Yaskawa INFORM job: DEMO_ROOF_SIDE_0625_3PAINT_26.JBI

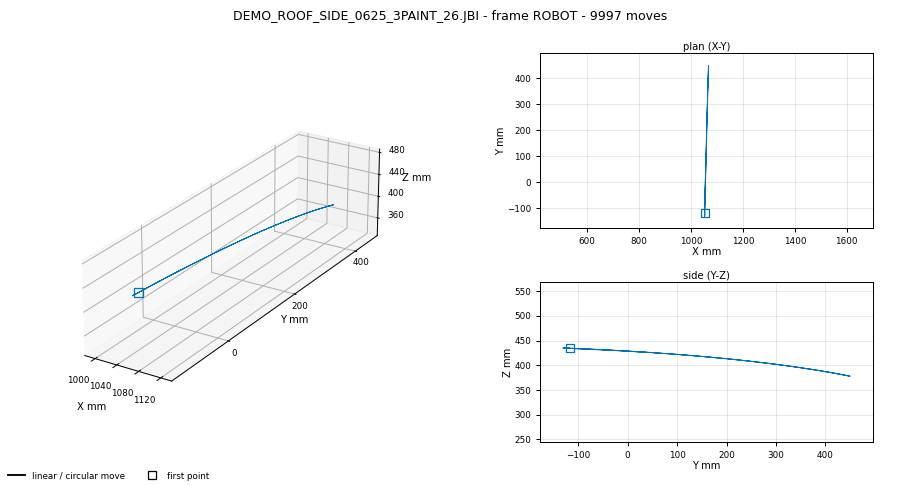
[picture p0: tool path of DEMO_ROOF_SIDE_0625_3PAINT_26.JBI in frame ROBOT, 9997 of 9997 moves have a stored position in this frame; points joined in program order, loops and branches not executed]
/JOB
//NAME DEMO_ROOF_SIDE_0625_3PAINT26
//POS
///NPOS 9997,0,0,0,0,0
///TOOL 0
///USER 0
///POSTYPE ROBOT
///RECTAN
///RCONF 1,0,0,0,0,0,0,0,0,0,0,0,0,0,0,0,0,0,0,0,0,0,0,0
C00000=1053.971,-116.920,435.028,170.360,28.855,155.473
C00001=1053.965,-117.170,435.037,170.358,28.855,155.473
C00002=1053.959,-117.419,435.047,170.356,28.854,155.473
C00003=1053.953,-117.669,435.057,170.354,28.853,155.473
C00004=1053.946,-117.919,435.066,170.352,28.853,155.473
C00005=1053.940,-118.169,435.076,170.349,28.852,155.473
C00006=1053.934,-118.419,435.084,170.347,28.852,155.474
C00007=1053.928,-118.669,435.094,170.345,28.851,155.474
C00008=1053.922,-118.918,435.103,170.343,28.851,155.474
C00009=1053.916,-119.168,435.112,170.341,28.850,155.474
C00010=1053.910,-119.417,435.122,170.339,28.850,155.474
C00011=1053.903,-119.667,435.131,170.337,28.849,155.474
C00012=1053.897,-119.917,435.141,170.335,28.849,155.474
C00013=1053.891,-120.167,435.151,170.333,28.848,155.474
C00014=1053.885,-120.417,435.160,170.331,28.847,155.474
C00015=1053.880,-120.666,435.169,170.329,28.847,155.474
C00016=1053.873,-120.916,435.178,170.327,28.847,155.474
C00017=1053.867,-121.166,435.187,170.324,28.846,155.474
C00018=1053.860,-121.415,435.197,170.322,28.846,155.474
C00019=1053.854,-121.665,435.206,170.320,28.845,155.475
C00020=1053.848,-121.915,435.216,170.319,28.845,155.475
C00021=1053.842,-122.165,435.225,170.317,28.844,155.475
C00022=1053.837,-122.414,435.234,170.315,28.844,155.475
C00023=1053.830,-122.664,435.243,170.312,28.843,155.475
C00024=1053.824,-122.914,435.252,170.310,28.843,155.475
C00025=1053.817,-123.164,435.262,170.308,28.842,155.475
C00026=1053.812,-123.414,435.271,170.306,28.842,155.475
C00027=1053.806,-123.663,435.280,170.304,28.842,155.475
C00028=1053.800,-123.913,435.290,170.302,28.841,155.475
C00029=1053.793,-124.162,435.299,170.299,28.841,155.475
C00030=1053.787,-124.413,435.307,170.297,28.840,155.476
C00031=1053.781,-124.663,435.317,170.295,28.840,155.476
C00032=1053.775,-124.912,435.326,170.294,28.840,155.476
C00033=1053.769,-125.162,435.334,170.292,28.839,155.476
C00034=1053.762,-125.412,435.344,170.290,28.839,155.476
C00035=1053.756,-125.661,435.354,170.287,28.838,155.476
C00036=1053.750,-125.911,435.363,170.285,28.838,155.476
C00037=1053.744,-126.161,435.371,170.283,28.838,155.476
C00038=1053.738,-126.410,435.381,170.281,28.838,155.476
C00039=1053.732,-126.660,435.390,170.279,28.837,155.477
C00040=1053.725,-126.910,435.398,170.276,28.837,155.477
C00041=1053.720,-127.159,435.408,170.274,28.836,155.477
C00042=1053.714,-127.410,435.417,170.272,28.836,155.477
C00043=1053.707,-127.659,435.425,170.271,28.835,155.477
C00044=1053.701,-127.909,435.436,170.269,28.835,155.477
C00045=1053.697,-128.159,435.445,170.267,28.835,155.477
C00046=1053.693,-128.409,435.455,170.265,28.833,155.477
C00047=1053.691,-128.659,435.466,170.263,28.831,155.477
C00048=1053.689,-128.909,435.479,170.262,28.828,155.476
C00049=1053.689,-129.161,435.491,170.260,28.825,155.476
C00050=1053.690,-129.411,435.503,170.259,28.822,155.475
C00051=1053.692,-129.660,435.518,170.258,28.818,155.475
C00052=1053.696,-129.912,435.532,170.257,28.813,155.474
C00053=1053.700,-130.163,435.547,170.256,28.808,155.473
C00054=1053.706,-130.413,435.563,170.256,28.802,155.472
C00055=1053.713,-130.663,435.580,170.256,28.796,155.471
C00056=1053.343,-130.687,435.365,170.208,28.964,155.504
C00057=1053.336,-130.437,435.348,170.208,28.970,155.505
C00058=1053.331,-130.186,435.333,170.209,28.975,155.506
C00059=1053.326,-129.936,435.318,170.210,28.981,155.507
C00060=1053.323,-129.684,435.303,170.210,28.985,155.508
C00061=1053.320,-129.434,435.290,170.212,28.989,155.508
C00062=1053.320,-129.183,435.276,170.213,28.993,155.509
C00063=1053.320,-128.933,435.264,170.214,28.996,155.509
C00064=1053.321,-128.683,435.251,170.216,28.998,155.510
C00065=1053.323,-128.432,435.240,170.218,29.001,155.510
C00066=1053.327,-128.182,435.230,170.219,29.002,155.510
C00067=1053.331,-127.932,435.220,170.221,29.003,155.510
C00068=1053.337,-127.682,435.211,170.223,29.004,155.510
C00069=1053.343,-127.433,435.202,170.225,29.004,155.510
C00070=1053.349,-127.183,435.193,170.227,29.004,155.510
C00071=1053.355,-126.933,435.184,170.230,29.004,155.510
C00072=1053.361,-126.683,435.174,170.232,29.005,155.509
C00073=1053.368,-126.434,435.166,170.234,29.005,155.509
C00074=1053.374,-126.184,435.157,170.236,29.006,155.509
C00075=1053.380,-125.934,435.147,170.237,29.006,155.509
C00076=1053.387,-125.685,435.138,170.240,29.006,155.509
C00077=1053.392,-125.435,435.130,170.242,29.006,155.509
C00078=1053.398,-125.185,435.120,170.244,29.007,155.509
C00079=1053.404,-124.935,435.111,170.246,29.007,155.509
C00080=1053.411,-124.686,435.102,170.248,29.008,155.509
C00081=1053.417,-124.435,435.093,170.251,29.008,155.509
C00082=1053.423,-124.186,435.084,170.253,29.009,155.508
C00083=1053.429,-123.937,435.074,170.255,29.009,155.508
C00084=1053.435,-123.686,435.066,170.257,29.010,155.508
C00085=1053.442,-123.437,435.056,170.259,29.010,155.508
C00086=1053.448,-123.187,435.047,170.261,29.010,155.508
C00087=1053.453,-122.938,435.037,170.264,29.010,155.508
C00088=1053.460,-122.688,435.028,170.265,29.011,155.508
C00089=1053.465,-122.438,435.019,170.267,29.011,155.508
C00090=1053.472,-122.188,435.010,170.269,29.012,155.508
C00091=1053.478,-121.938,435.000,170.271,29.012,155.508
C00092=1053.485,-121.688,434.991,170.273,29.012,155.507
C00093=1053.490,-121.439,434.982,170.276,29.013,155.507
C00094=1053.496,-121.189,434.973,170.278,29.013,155.507
C00095=1053.502,-120.939,434.963,170.280,29.014,155.507
C00096=1053.508,-120.689,434.954,170.282,29.014,155.507
C00097=1053.515,-120.440,434.945,170.284,29.015,155.507
C00098=1053.522,-120.190,434.935,170.285,29.016,155.507
C00099=1053.528,-119.940,434.926,170.288,29.016,155.507
C00100=1053.533,-119.691,434.916,170.290,29.017,155.507
C00101=1053.539,-119.441,434.908,170.292,29.017,155.507
C00102=1053.545,-119.191,434.898,170.294,29.018,155.507
C00103=1053.551,-118.941,434.888,170.296,29.018,155.507
C00104=1053.558,-118.691,434.879,170.299,29.019,155.507
C00105=1053.564,-118.442,434.869,170.301,29.019,155.506
C00106=1053.570,-118.192,434.860,170.303,29.019,155.506
C00107=1053.577,-117.942,434.851,170.305,29.020,155.506
C00108=1053.582,-117.693,434.842,170.307,29.020,155.506
C00109=1053.589,-117.443,434.832,170.308,29.021,155.506
C00110=1053.595,-117.194,434.822,170.311,29.022,155.506
C00111=1053.601,-116.944,434.813,170.313,29.022,155.506
C00112=1053.607,-116.694,434.803,170.315,29.023,155.506
C00113=1053.613,-116.444,434.794,170.317,29.023,155.506
C00114=1053.620,-116.194,434.784,170.319,29.024,155.506
C00115=1053.626,-115.945,434.775,170.321,29.024,155.506
C00116=1053.632,-115.695,434.765,170.324,29.025,155.506
C00117=1053.638,-115.411,434.755,170.326,29.026,155.506
C00118=1053.646,-115.126,434.743,170.328,29.026,155.505
C00119=1053.653,-114.841,434.733,170.330,29.027,155.505
C00120=1053.660,-114.558,434.722,170.332,29.027,155.505
C00121=1053.666,-114.308,434.712,170.335,29.028,155.505
C00122=1053.672,-114.058,434.703,170.337,29.029,155.505
C00123=1053.678,-113.808,434.693,170.339,29.029,155.505
C00124=1053.684,-113.558,434.683,170.341,29.030,155.505
C00125=1053.690,-113.308,434.673,170.343,29.031,155.505
C00126=1053.696,-113.059,434.664,170.345,29.031,155.505
C00127=1053.702,-112.809,434.654,170.348,29.032,155.505
C00128=1053.709,-112.559,434.645,170.349,29.033,155.505
C00129=1053.715,-112.309,434.635,170.351,29.033,155.505
C00130=1053.721,-112.059,434.626,170.353,29.033,155.505
C00131=1053.727,-111.810,434.615,170.355,29.034,155.505
C00132=1053.734,-111.560,434.606,170.357,29.035,155.505
C00133=1053.740,-111.311,434.596,170.360,29.035,155.505
C00134=1053.746,-111.061,434.587,170.362,29.037,155.505
C00135=1053.751,-110.811,434.576,170.364,29.037,155.505
C00136=1053.757,-110.561,434.567,170.366,29.037,155.504
C00137=1053.764,-110.312,434.557,170.367,29.038,155.505
C00138=1053.770,-110.062,434.547,170.369,29.039,155.504
C00139=1053.776,-109.812,434.537,170.372,29.039,155.504
C00140=1053.782,-109.562,434.528,170.374,29.040,155.504
C00141=1053.789,-109.313,434.518,170.376,29.041,155.504
C00142=1053.795,-109.063,434.508,170.378,29.041,155.504
C00143=1053.801,-108.814,434.498,170.380,29.042,155.504
C00144=1053.807,-108.563,434.488,170.382,29.043,155.504
C00145=1053.813,-108.314,434.479,170.384,29.044,155.504
C00146=1053.819,-108.064,434.469,170.386,29.044,155.504
C00147=1053.826,-107.815,434.459,170.388,29.045,155.504
C00148=1053.832,-107.565,434.449,170.390,29.046,155.504
C00149=1053.838,-107.315,434.440,170.392,29.046,155.504
C00150=1053.844,-107.066,434.429,170.394,29.047,155.504
C00151=1053.850,-106.816,434.419,170.397,29.048,155.504
C00152=1053.856,-106.566,434.410,170.399,29.049,155.504
C00153=1053.862,-106.316,434.400,170.400,29.049,155.504
C00154=1053.869,-106.066,434.389,170.402,29.050,155.504
C00155=1053.875,-105.816,434.379,170.404,29.051,155.504
C00156=1053.881,-105.566,434.370,170.406,29.052,155.504
C00157=1053.887,-105.317,434.359,170.409,29.052,155.504
C00158=1053.893,-105.067,434.349,170.411,29.053,155.504
C00159=1053.899,-104.817,434.340,170.413,29.054,155.504
C00160=1053.905,-104.568,434.329,170.415,29.055,155.504
C00161=1053.912,-104.318,434.320,170.416,29.056,155.504
C00162=1053.917,-104.069,434.309,170.418,29.056,155.504
C00163=1053.923,-103.819,434.299,170.420,29.057,155.504
C00164=1053.930,-103.569,434.290,170.423,29.058,155.504
C00165=1053.936,-103.319,434.279,170.425,29.059,155.504
C00166=1053.942,-103.069,434.269,170.427,29.060,155.504
C00167=1053.949,-102.820,434.259,170.429,29.060,155.504
C00168=1053.954,-102.570,434.249,170.431,29.061,155.504
C00169=1053.960,-102.320,434.239,170.432,29.062,155.503
C00170=1053.967,-102.071,434.229,170.434,29.063,155.503
C00171=1053.972,-101.821,434.219,170.437,29.064,155.503
C00172=1053.979,-101.572,434.208,170.439,29.064,155.503
C00173=1053.985,-101.321,434.198,170.441,29.065,155.503
C00174=1053.991,-101.072,434.188,170.443,29.066,155.503
C00175=1053.997,-100.822,434.178,170.445,29.067,155.503
C00176=1054.004,-100.573,434.168,170.446,29.068,155.503
C00177=1054.009,-100.323,434.158,170.449,29.069,155.503
C00178=1054.016,-100.073,434.147,170.451,29.069,155.503
C00179=1054.022,-99.823,434.137,170.453,29.070,155.503
C00180=1054.028,-99.573,434.126,170.455,29.072,155.503
C00181=1054.035,-99.287,434.115,170.457,29.072,155.503
C00182=1054.042,-99.001,434.103,170.460,29.073,155.503
C00183=1054.050,-98.716,434.092,170.461,29.074,155.503
C00184=1054.057,-98.431,434.080,170.464,29.075,155.503
C00185=1054.063,-98.180,434.070,170.466,29.076,155.503
C00186=1054.069,-97.931,434.060,170.468,29.077,155.503
C00187=1054.075,-97.682,434.049,170.470,29.078,155.503
C00188=1054.081,-97.432,434.039,170.472,29.079,155.503
C00189=1054.087,-97.182,434.028,170.475,29.079,155.503
C00190=1054.094,-96.932,434.018,170.476,29.080,155.503
C00191=1054.099,-96.682,434.007,170.478,29.082,155.503
C00192=1054.106,-96.433,433.997,170.480,29.083,155.503
C00193=1054.111,-96.183,433.987,170.482,29.084,155.503
C00194=1054.118,-95.934,433.977,170.484,29.085,155.503
C00195=1054.124,-95.684,433.965,170.486,29.086,155.503
C00196=1054.130,-95.434,433.955,170.488,29.087,155.504
C00197=1054.136,-95.184,433.945,170.490,29.088,155.503
C00198=1054.142,-94.935,433.934,170.492,29.088,155.503
C00199=1054.148,-94.685,433.925,170.494,29.089,155.503
C00200=1054.154,-94.435,433.913,170.496,29.090,155.503
C00201=1054.160,-94.186,433.902,170.498,29.091,155.504
C00202=1054.167,-93.936,433.892,170.500,29.092,155.504
C00203=1054.172,-93.686,433.882,170.502,29.093,155.504
C00204=1054.179,-93.436,433.871,170.504,29.095,155.504
C00205=1054.185,-93.187,433.860,170.506,29.096,155.504
C00206=1054.190,-92.937,433.850,170.508,29.097,155.504
C00207=1054.197,-92.688,433.840,170.510,29.098,155.504
C00208=1054.203,-92.437,433.829,170.512,29.099,155.504
C00209=1054.209,-92.188,433.818,170.514,29.100,155.504
C00210=1054.215,-91.939,433.808,170.515,29.101,155.504
C00211=1054.221,-91.689,433.797,170.517,29.102,155.504
C00212=1054.228,-91.439,433.787,170.520,29.103,155.504
C00213=1054.233,-91.189,433.776,170.522,29.104,155.504
C00214=1054.239,-90.940,433.765,170.524,29.105,155.504
C00215=1054.246,-90.690,433.754,170.526,29.106,155.504
C00216=1054.252,-90.440,433.744,170.527,29.107,155.504
C00217=1054.257,-90.190,433.733,170.529,29.108,155.504
C00218=1054.264,-89.941,433.723,170.531,29.109,155.504
C00219=1054.270,-89.691,433.712,170.533,29.110,155.504
C00220=1054.276,-89.441,433.701,170.536,29.111,155.504
C00221=1054.282,-89.192,433.691,170.538,29.112,155.504
C00222=1054.289,-88.942,433.679,170.540,29.113,155.504
C00223=1054.295,-88.692,433.670,170.541,29.114,155.504
C00224=1054.301,-88.443,433.659,170.543,29.115,155.504
C00225=1054.307,-88.193,433.648,170.545,29.116,155.504
C00226=1054.314,-87.943,433.637,170.547,29.117,155.504
C00227=1054.319,-87.694,433.627,170.549,29.118,155.504
C00228=1054.326,-87.444,433.615,170.552,29.120,155.504
C00229=1054.332,-87.195,433.605,170.553,29.121,155.504
C00230=1054.338,-86.944,433.594,170.555,29.122,155.504
C00231=1054.344,-86.695,433.583,170.557,29.123,155.504
C00232=1054.351,-86.446,433.573,170.559,29.124,155.504
C00233=1054.357,-86.195,433.561,170.561,29.125,155.504
C00234=1054.363,-85.946,433.550,170.563,29.126,155.505
C00235=1054.369,-85.696,433.540,170.565,29.127,155.505
C00236=1054.376,-85.447,433.529,170.567,29.129,155.505
C00237=1054.381,-85.197,433.518,170.569,29.130,155.505
C00238=1054.388,-84.947,433.507,170.571,29.131,155.505
C00239=1054.394,-84.698,433.497,170.573,29.132,155.505
C00240=1054.400,-84.448,433.485,170.575,29.133,155.505
C00241=1054.406,-84.198,433.474,170.577,29.134,155.505
C00242=1054.413,-83.949,433.464,170.578,29.135,155.505
C00243=1054.419,-83.699,433.453,170.580,29.136,155.505
C00244=1054.425,-83.449,433.442,170.583,29.137,155.505
C00245=1054.432,-83.165,433.429,170.585,29.139,155.505
C00246=1054.439,-82.882,433.418,170.587,29.140,155.505
C00247=1054.446,-82.598,433.405,170.589,29.141,155.505
C00248=1054.454,-82.315,433.392,170.591,29.142,155.505
C00249=1054.460,-82.066,433.381,170.593,29.143,155.505
C00250=1054.466,-81.815,433.370,170.595,29.144,155.505
C00251=1054.472,-81.566,433.359,170.597,29.145,155.505
C00252=1054.479,-81.316,433.349,170.600,29.147,155.505
C00253=1054.485,-81.067,433.338,170.601,29.148,155.505
C00254=1054.491,-80.816,433.327,170.603,29.149,155.506
C00255=1054.497,-80.567,433.316,170.605,29.150,155.506
C00256=1054.504,-80.317,433.305,170.607,29.151,155.506
C00257=1054.510,-80.068,433.293,170.609,29.152,155.506
C00258=1054.516,-79.818,433.282,170.611,29.153,155.506
C00259=1054.522,-79.568,433.271,170.612,29.155,155.506
C00260=1054.528,-79.318,433.260,170.614,29.156,155.506
C00261=1054.534,-79.069,433.249,170.617,29.157,155.506
C00262=1054.540,-78.820,433.238,170.619,29.159,155.506
C00263=1054.546,-78.570,433.226,170.621,29.160,155.506
C00264=1054.552,-78.320,433.215,170.623,29.161,155.506
C00265=1054.559,-78.070,433.205,170.624,29.162,155.506
C00266=1054.565,-77.821,433.193,170.626,29.163,155.506
C00267=1054.572,-77.571,433.182,170.628,29.165,155.506
C00268=1054.577,-77.322,433.171,170.630,29.166,155.506
C00269=1054.584,-77.072,433.160,170.632,29.167,155.506
C00270=1054.590,-76.823,433.148,170.633,29.169,155.507
C00271=1054.596,-76.573,433.137,170.636,29.170,155.507
C00272=1054.602,-76.323,433.126,170.638,29.172,155.507
C00273=1054.608,-76.073,433.115,170.640,29.173,155.507
C00274=1054.615,-75.823,433.103,170.642,29.174,155.507
C00275=1054.621,-75.574,433.092,170.644,29.175,155.507
C00276=1054.627,-75.324,433.081,170.645,29.176,155.507
C00277=1054.633,-75.075,433.069,170.647,29.178,155.507
C00278=1054.639,-74.825,433.058,170.649,29.179,155.507
C00279=1054.645,-74.575,433.047,170.651,29.180,155.507
C00280=1054.652,-74.325,433.035,170.653,29.182,155.507
C00281=1054.657,-74.076,433.024,170.656,29.183,155.507
C00282=1054.664,-73.826,433.012,170.657,29.184,155.508
C00283=1054.670,-73.577,433.001,170.659,29.185,155.508
C00284=1054.675,-73.326,432.990,170.661,29.187,155.508
C00285=1054.682,-73.077,432.978,170.663,29.189,155.508
C00286=1054.688,-72.827,432.967,170.665,29.190,155.508
C00287=1054.694,-72.578,432.955,170.666,29.191,155.508
C00288=1054.700,-72.328,432.944,170.668,29.192,155.508
C00289=1054.706,-72.078,432.932,170.670,29.194,155.508
C00290=1054.712,-71.829,432.920,170.672,29.195,155.508
C00291=1054.718,-71.579,432.909,170.674,29.196,155.508
C00292=1054.724,-71.330,432.898,170.675,29.198,155.509
C00293=1054.730,-71.079,432.886,170.677,29.199,155.509
C00294=1054.736,-70.830,432.874,170.679,29.201,155.509
C00295=1054.742,-70.580,432.863,170.682,29.203,155.509
C00296=1054.749,-70.331,432.851,170.684,29.204,155.509
C00297=1054.754,-70.081,432.840,170.685,29.205,155.509
C00298=1054.761,-69.831,432.828,170.687,29.207,155.509
C00299=1054.766,-69.582,432.817,170.689,29.208,155.509
C00300=1054.773,-69.332,432.805,170.691,29.209,155.509
C00301=1054.778,-69.082,432.793,170.693,29.211,155.510
C00302=1054.785,-68.833,432.781,170.695,29.212,155.510
C00303=1054.791,-68.583,432.769,170.696,29.214,155.510
C00304=1054.797,-68.334,432.758,170.698,29.215,155.510
C00305=1054.803,-68.084,432.746,170.700,29.216,155.510
C00306=1054.809,-67.834,432.735,170.702,29.218,155.510
C00307=1054.815,-67.585,432.723,170.704,29.220,155.510
C00308=1054.822,-67.335,432.712,170.705,29.221,155.510
C00309=1054.828,-67.054,432.698,170.708,29.222,155.510
C00310=1054.835,-66.773,432.684,170.710,29.224,155.511
C00311=1054.842,-66.492,432.672,170.712,29.226,155.511
C00312=1054.849,-66.210,432.658,170.714,29.227,155.511
C00313=1054.855,-65.960,432.647,170.716,29.229,155.511
C00314=1054.861,-65.711,432.635,170.718,29.230,155.511
C00315=1054.867,-65.461,432.623,170.720,29.232,155.511
C00316=1054.873,-65.211,432.612,170.722,29.233,155.511
C00317=1054.880,-64.962,432.600,170.723,29.235,155.511
C00318=1054.886,-64.712,432.587,170.725,29.236,155.511
C00319=1054.891,-64.462,432.576,170.727,29.238,155.512
C00320=1054.898,-64.213,432.564,170.729,29.239,155.512
C00321=1054.905,-63.963,432.552,170.731,29.241,155.512
C00322=1054.910,-63.713,432.541,170.732,29.242,155.512
C00323=1054.916,-63.464,432.529,170.734,29.243,155.512
C00324=1054.923,-63.214,432.517,170.736,29.245,155.512
C00325=1054.929,-62.964,432.504,170.739,29.247,155.512
C00326=1054.935,-62.715,432.494,170.741,29.248,155.512
C00327=1054.941,-62.465,432.482,170.742,29.249,155.513
C00328=1054.947,-62.215,432.469,170.744,29.251,155.513
C00329=1054.954,-61.966,432.457,170.746,29.253,155.513
C00330=1054.960,-61.716,432.446,170.748,29.254,155.513
C00331=1054.965,-61.466,432.434,170.750,29.255,155.513
C00332=1054.972,-61.217,432.422,170.751,29.257,155.513
C00333=1054.979,-60.967,432.410,170.753,29.259,155.513
C00334=1054.984,-60.718,432.398,170.755,29.260,155.514
C00335=1054.990,-60.468,432.386,170.757,29.261,155.514
C00336=1054.997,-60.218,432.374,170.759,29.263,155.514
C00337=1055.003,-59.968,432.362,170.760,29.264,155.514
C00338=1055.009,-59.720,432.350,170.762,29.266,155.514
C00339=1055.016,-59.470,432.338,170.764,29.268,155.514
C00340=1055.022,-59.220,432.326,170.766,29.269,155.514
C00341=1055.028,-58.970,432.314,170.768,29.270,155.514
C00342=1055.035,-58.720,432.302,170.769,29.272,155.515
C00343=1055.040,-58.471,432.290,170.772,29.274,155.515
C00344=1055.046,-58.222,432.278,170.774,29.275,155.515
C00345=1055.052,-57.972,432.266,170.776,29.277,155.515
C00346=1055.059,-57.722,432.254,170.778,29.278,155.515
C00347=1055.066,-57.473,432.242,170.779,29.279,155.515
C00348=1055.072,-57.223,432.229,170.781,29.281,155.515
C00349=1055.078,-56.974,432.218,170.783,29.283,155.515
C00350=1055.084,-56.724,432.206,170.785,29.284,155.516
C00351=1055.090,-56.474,432.193,170.787,29.286,155.516
C00352=1055.097,-56.224,432.182,170.788,29.287,155.516
C00353=1055.102,-55.974,432.169,170.790,29.289,155.516
C00354=1055.109,-55.725,432.157,170.792,29.290,155.516
C00355=1055.116,-55.475,432.145,170.794,29.292,155.516
C00356=1055.122,-55.225,432.133,170.796,29.293,155.516
C00357=1055.128,-54.976,432.121,170.797,29.295,155.517
C00358=1055.134,-54.726,432.109,170.799,29.297,155.517
C00359=1055.140,-54.477,432.097,170.801,29.298,155.517
C00360=1055.147,-54.227,432.085,170.803,29.299,155.517
C00361=1055.153,-53.977,432.072,170.805,29.301,155.517
C00362=1055.159,-53.728,432.060,170.806,29.302,155.517
C00363=1055.165,-53.478,432.048,170.808,29.304,155.517
C00364=1055.172,-53.228,432.036,170.810,29.306,155.517
C00365=1055.179,-52.979,432.024,170.812,29.307,155.518
C00366=1055.185,-52.730,432.011,170.814,29.309,155.518
C00367=1055.192,-52.480,431.999,170.815,29.310,155.518
C00368=1055.197,-52.231,431.986,170.818,29.312,155.518
C00369=1055.203,-51.981,431.975,170.820,29.314,155.518
C00370=1055.209,-51.731,431.962,170.822,29.315,155.518
C00371=1055.216,-51.482,431.950,170.824,29.316,155.518
C00372=1055.223,-51.232,431.938,170.825,29.318,155.519
C00373=1055.229,-50.952,431.924,170.827,29.320,155.519
C00374=1055.237,-50.672,431.910,170.829,29.322,155.519
C00375=1055.244,-50.392,431.897,170.831,29.324,155.519
C00376=1055.251,-50.112,431.882,170.833,29.325,155.519
C00377=1055.257,-49.862,431.869,170.835,29.327,155.519
C00378=1055.263,-49.612,431.857,170.837,29.329,155.520
C00379=1055.269,-49.363,431.845,170.839,29.331,155.520
C00380=1055.275,-49.113,431.833,170.841,29.332,155.520
C00381=1055.281,-48.864,431.820,170.842,29.334,155.520
C00382=1055.287,-48.614,431.807,170.844,29.336,155.520
C00383=1055.294,-48.365,431.795,170.846,29.337,155.520
C00384=1055.300,-48.115,431.782,170.848,29.339,155.521
C00385=1055.306,-47.865,431.770,170.849,29.341,155.521
C00386=1055.312,-47.616,431.756,170.851,29.343,155.521
C00387=1055.318,-47.366,431.745,170.853,29.344,155.521
C00388=1055.324,-47.116,431.732,170.855,29.346,155.521
C00389=1055.330,-46.866,431.719,170.857,29.347,155.521
C00390=1055.336,-46.617,431.706,170.858,29.349,155.522
C00391=1055.343,-46.368,431.694,170.860,29.351,155.522
C00392=1055.349,-46.118,431.682,170.862,29.353,155.522
C00393=1055.355,-45.868,431.668,170.864,29.354,155.522
C00394=1055.361,-45.619,431.656,170.866,29.356,155.522
C00395=1055.368,-45.369,431.644,170.867,29.358,155.522
C00396=1055.374,-45.120,431.631,170.869,29.360,155.523
C00397=1055.380,-44.870,431.618,170.871,29.361,155.523
C00398=1055.386,-44.620,431.605,170.873,29.363,155.523
C00399=1055.393,-44.371,431.593,170.874,29.365,155.523
C00400=1055.399,-44.121,431.580,170.876,29.366,155.523
C00401=1055.405,-43.871,431.568,170.878,29.369,155.524
C00402=1055.411,-43.622,431.554,170.880,29.370,155.524
C00403=1055.417,-43.372,431.542,170.882,29.372,155.524
C00404=1055.423,-43.122,431.530,170.883,29.373,155.524
C00405=1055.430,-42.873,431.517,170.885,29.376,155.524
C00406=1055.435,-42.623,431.504,170.887,29.377,155.525
C00407=1055.442,-42.374,431.491,170.889,29.379,155.525
C00408=1055.448,-42.124,431.478,170.890,29.380,155.525
C00409=1055.455,-41.875,431.466,170.892,29.382,155.525
C00410=1055.460,-41.625,431.453,170.894,29.384,155.525
C00411=1055.466,-41.375,431.440,170.896,29.386,155.525
C00412=1055.473,-41.126,431.427,170.898,29.387,155.526
C00413=1055.478,-40.876,431.415,170.899,29.389,155.526
C00414=1055.485,-40.627,431.402,170.901,29.391,155.526
C00415=1055.491,-40.377,431.389,170.903,29.393,155.526
C00416=1055.498,-40.128,431.376,170.905,29.394,155.526
C00417=1055.503,-39.878,431.364,170.906,29.396,155.526
C00418=1055.510,-39.628,431.350,170.908,29.398,155.527
C00419=1055.516,-39.378,431.337,170.910,29.400,155.527
C00420=1055.523,-39.130,431.325,170.912,29.401,155.527
C00421=1055.529,-38.880,431.312,170.914,29.404,155.527
C00422=1055.535,-38.630,431.299,170.915,29.405,155.527
C00423=1055.541,-38.380,431.286,170.917,29.407,155.528
C00424=1055.547,-38.131,431.273,170.919,29.409,155.528
C00425=1055.553,-37.881,431.261,170.921,29.411,155.528
C00426=1055.560,-37.632,431.247,170.922,29.412,155.528
C00427=1055.566,-37.383,431.234,170.923,29.414,155.528
C00428=1055.572,-37.133,431.221,170.925,29.416,155.529
C00429=1055.578,-36.883,431.208,170.927,29.418,155.529
C00430=1055.584,-36.633,431.195,170.929,29.420,155.529
C00431=1055.591,-36.384,431.182,170.930,29.422,155.529
C00432=1055.596,-36.134,431.168,170.932,29.423,155.529
C00433=1055.602,-35.884,431.156,170.934,29.425,155.530
C00434=1055.608,-35.635,431.142,170.936,29.427,155.530
C00435=1055.614,-35.386,431.129,170.937,29.429,155.530
C00436=1055.620,-35.136,431.116,170.939,29.431,155.530
C00437=1055.627,-34.856,431.102,170.941,29.433,155.530
C00438=1055.634,-34.577,431.087,170.944,29.435,155.531
C00439=1055.641,-34.297,431.072,170.945,29.437,155.531
C00440=1055.648,-34.018,431.058,170.947,29.439,155.531
C00441=1055.654,-33.768,431.044,170.949,29.441,155.531
C00442=1055.660,-33.518,431.031,170.951,29.443,155.532
C00443=1055.667,-33.269,431.018,170.952,29.445,155.532
C00444=1055.673,-33.019,431.005,170.954,29.446,155.532
C00445=1055.679,-32.770,430.991,170.956,29.449,155.532
C00446=1055.685,-32.520,430.979,170.958,29.450,155.532
C00447=1055.692,-32.270,430.965,170.960,29.452,155.533
C00448=1055.698,-32.021,430.952,170.961,29.454,155.533
C00449=1055.704,-31.772,430.939,170.963,29.456,155.533
C00450=1055.710,-31.522,430.926,170.965,29.458,155.533
C00451=1055.716,-31.273,430.913,170.966,29.460,155.534
C00452=1055.723,-31.023,430.899,170.967,29.461,155.534
C00453=1055.729,-30.773,430.885,170.969,29.464,155.534
C00454=1055.735,-30.524,430.872,170.971,29.465,155.534
C00455=1055.741,-30.274,430.860,170.973,29.467,155.534
C00456=1055.748,-30.024,430.846,170.975,29.469,155.535
C00457=1055.754,-29.775,430.833,170.976,29.471,155.535
C00458=1055.760,-29.525,430.819,170.978,29.473,155.535
C00459=1055.766,-29.276,430.806,170.980,29.475,155.535
C00460=1055.772,-29.027,430.793,170.982,29.477,155.535
C00461=1055.779,-28.776,430.780,170.983,29.479,155.536
C00462=1055.784,-28.527,430.766,170.985,29.480,155.536
C00463=1055.791,-28.277,430.753,170.987,29.483,155.536
C00464=1055.797,-28.027,430.739,170.989,29.484,155.536
C00465=1055.804,-27.778,430.726,170.990,29.486,155.537
C00466=1055.810,-27.529,430.713,170.992,29.488,155.537
C00467=1055.816,-27.280,430.699,170.994,29.490,155.537
C00468=1055.823,-27.030,430.686,170.996,29.492,155.537
C00469=1055.828,-26.780,430.672,170.997,29.494,155.537
C00470=1055.835,-26.531,430.659,170.998,29.495,155.538
C00471=1055.840,-26.281,430.646,171.000,29.498,155.538
C00472=1055.847,-26.031,430.632,171.002,29.500,155.538
C00473=1055.853,-25.781,430.618,171.004,29.501,155.538
C00474=1055.859,-25.532,430.605,171.005,29.504,155.539
C00475=1055.864,-25.283,430.591,171.007,29.506,155.539
C00476=1055.871,-25.033,430.578,171.009,29.507,155.539
C00477=1055.877,-24.783,430.564,171.011,29.509,155.539
C00478=1055.883,-24.534,430.551,171.012,29.512,155.540
C00479=1055.890,-24.284,430.537,171.014,29.513,155.540
C00480=1055.896,-24.035,430.524,171.016,29.515,155.540
C00481=1055.901,-23.785,430.510,171.018,29.518,155.540
C00482=1055.908,-23.536,430.497,171.019,29.519,155.540
C00483=1055.915,-23.286,430.482,171.020,29.521,155.541
C00484=1055.920,-23.037,430.468,171.022,29.523,155.541
C00485=1055.926,-22.788,430.455,171.024,29.525,155.541
C00486=1055.933,-22.537,430.441,171.026,29.527,155.541
C00487=1055.939,-22.288,430.428,171.027,29.529,155.542
C00488=1055.945,-22.039,430.414,171.029,29.531,155.542
C00489=1055.951,-21.788,430.400,171.031,29.533,155.542
C00490=1055.957,-21.539,430.387,171.033,29.535,155.542
C00491=1055.963,-21.290,430.374,171.034,29.537,155.543
C00492=1055.970,-21.040,430.359,171.036,29.539,155.543
C00493=1055.976,-20.790,430.346,171.038,29.541,155.543
C00494=1055.982,-20.541,430.331,171.040,29.544,155.543
C00495=1055.988,-20.291,430.318,171.040,29.545,155.544
C00496=1055.995,-20.042,430.305,171.042,29.547,155.544
C00497=1056.000,-19.793,430.291,171.044,29.549,155.544
C00498=1056.007,-19.543,430.277,171.046,29.551,155.544
C00499=1056.012,-19.293,430.263,171.047,29.553,155.545
C00500=1056.019,-19.044,430.249,171.049,29.555,155.545
C00501=1056.026,-18.763,430.233,171.051,29.558,155.545
C00502=1056.033,-18.483,430.219,171.053,29.560,155.545
C00503=1056.040,-18.202,430.203,171.054,29.562,155.546
C00504=1056.047,-17.923,430.187,171.057,29.564,155.546
C00505=1056.053,-17.672,430.173,171.058,29.566,155.546
C00506=1056.059,-17.423,430.160,171.060,29.568,155.546
C00507=1056.065,-17.174,430.145,171.061,29.570,155.547
C00508=1056.072,-16.924,430.132,171.063,29.572,155.547
C00509=1056.078,-16.675,430.118,171.065,29.574,155.547
C00510=1056.084,-16.425,430.104,171.067,29.576,155.547
C00511=1056.091,-16.176,430.090,171.069,29.578,155.548
C00512=1056.097,-15.926,430.076,171.070,29.580,155.548
C00513=1056.103,-15.676,430.063,171.072,29.582,155.548
C00514=1056.109,-15.427,430.049,171.074,29.584,155.548
C00515=1056.116,-15.178,430.035,171.075,29.586,155.549
C00516=1056.121,-14.928,430.021,171.076,29.588,155.549
C00517=1056.128,-14.678,430.007,171.078,29.591,155.549
C00518=1056.134,-14.429,429.992,171.080,29.593,155.549
C00519=1056.140,-14.179,429.978,171.082,29.594,155.550
C00520=1056.146,-13.930,429.965,171.083,29.596,155.550
C00521=1056.152,-13.681,429.950,171.085,29.599,155.550
C00522=1056.158,-13.430,429.936,171.087,29.601,155.550
C00523=1056.165,-13.182,429.922,171.089,29.603,155.551
C00524=1056.171,-12.931,429.908,171.089,29.605,155.551
C00525=1056.176,-12.682,429.894,171.091,29.607,155.551
C00526=1056.183,-12.432,429.880,171.093,29.609,155.551
C00527=1056.189,-12.183,429.866,171.095,29.611,155.552
C00528=1056.194,-11.934,429.851,171.096,29.613,155.552
C00529=1056.201,-11.684,429.838,171.098,29.615,155.552
C00530=1056.207,-11.434,429.824,171.100,29.618,155.552
C00531=1056.213,-11.185,429.809,171.102,29.620,155.553
C00532=1056.219,-10.935,429.796,171.103,29.622,155.553
C00533=1056.226,-10.686,429.781,171.104,29.624,155.553
C00534=1056.231,-10.436,429.767,171.106,29.626,155.554
C00535=1056.238,-10.187,429.752,171.108,29.628,155.554
C00536=1056.244,-9.937,429.739,171.110,29.630,155.554
C00537=1056.250,-9.688,429.724,171.111,29.632,155.554
C00538=1056.256,-9.438,429.710,171.113,29.634,155.555
C00539=1056.263,-9.189,429.695,171.115,29.636,155.555
C00540=1056.268,-8.939,429.681,171.116,29.638,155.555
C00541=1056.275,-8.690,429.667,171.117,29.641,155.555
C00542=1056.281,-8.440,429.653,171.119,29.643,155.556
C00543=1056.287,-8.191,429.638,171.121,29.645,155.556
C00544=1056.293,-7.941,429.625,171.123,29.647,155.556
C00545=1056.300,-7.692,429.610,171.124,29.649,155.556
C00546=1056.306,-7.441,429.596,171.126,29.651,155.557
C00547=1056.312,-7.192,429.581,171.128,29.653,155.557
C00548=1056.319,-6.943,429.567,171.129,29.655,155.557
C00549=1056.324,-6.693,429.553,171.130,29.657,155.558
C00550=1056.331,-6.444,429.538,171.132,29.659,155.558
C00551=1056.337,-6.195,429.525,171.134,29.662,155.558
C00552=1056.343,-5.945,429.510,171.136,29.664,155.558
C00553=1056.349,-5.696,429.495,171.137,29.666,155.559
C00554=1056.355,-5.446,429.481,171.139,29.668,155.559
C00555=1056.362,-5.196,429.467,171.140,29.670,155.559
C00556=1056.368,-4.947,429.452,171.142,29.672,155.559
C00557=1056.374,-4.697,429.438,171.144,29.674,155.560
C00558=1056.381,-4.448,429.424,171.145,29.676,155.560
C00559=1056.387,-4.198,429.410,171.147,29.678,155.560
C00560=1056.393,-3.949,429.395,171.149,29.680,155.560
C00561=1056.399,-3.700,429.380,171.151,29.683,155.561
C00562=1056.406,-3.450,429.366,171.152,29.685,155.561
C00563=1056.411,-3.201,429.352,171.153,29.687,155.561
C00564=1056.418,-2.951,429.337,171.155,29.689,155.562
C00565=1056.425,-2.669,429.320,171.157,29.692,155.562
C00566=1056.431,-2.387,429.304,171.158,29.694,155.562
C00567=1056.438,-2.105,429.287,171.160,29.697,155.563
C00568=1056.444,-1.823,429.271,171.163,29.699,155.563
C00569=1056.451,-1.574,429.256,171.164,29.701,155.563
C00570=1056.457,-1.323,429.241,171.165,29.703,155.563
C00571=1056.463,-1.074,429.227,171.167,29.705,155.564
C00572=1056.469,-0.825,429.212,171.169,29.708,155.564
C00573=1056.475,-0.576,429.197,171.170,29.710,155.564
C00574=1056.481,-0.326,429.182,171.172,29.713,155.565
C00575=1056.487,-0.076,429.169,171.173,29.715,155.565
C00576=1056.493,0.173,429.154,171.175,29.717,155.565
C00577=1056.499,0.423,429.139,171.177,29.719,155.566
C00578=1056.505,0.672,429.124,171.178,29.721,155.566
C00579=1056.512,0.922,429.109,171.180,29.723,155.566
C00580=1056.518,1.171,429.094,171.182,29.725,155.566
C00581=1056.523,1.421,429.080,171.183,29.727,155.567
C00582=1056.530,1.670,429.065,171.184,29.730,155.567
C00583=1056.536,1.919,429.051,171.186,29.732,155.567
C00584=1056.542,2.169,429.036,171.188,29.735,155.568
C00585=1056.548,2.419,429.021,171.190,29.737,155.568
C00586=1056.554,2.668,429.006,171.191,29.739,155.568
C00587=1056.561,2.917,428.991,171.192,29.741,155.568
C00588=1056.567,3.167,428.976,171.194,29.743,155.569
C00589=1056.573,3.416,428.962,171.196,29.745,155.569
C00590=1056.579,3.666,428.947,171.197,29.748,155.569
C00591=1056.585,3.916,428.933,171.199,29.750,155.570
C00592=1056.591,4.165,428.918,171.200,29.752,155.570
C00593=1056.597,4.415,428.903,171.202,29.754,155.570
C00594=1056.603,4.664,428.888,171.203,29.756,155.571
C00595=1056.609,4.913,428.873,171.205,29.759,155.571
C00596=1056.615,5.163,428.858,171.207,29.761,155.571
C00597=1056.622,5.413,428.843,171.209,29.763,155.571
C00598=1056.628,5.662,428.828,171.209,29.765,155.572
C00599=1056.634,5.911,428.814,171.211,29.768,155.572
C00600=1056.640,6.161,428.799,171.213,29.770,155.572
C00601=1056.646,6.411,428.784,171.215,29.772,155.573
C00602=1056.653,6.660,428.769,171.216,29.774,155.573
C00603=1056.659,6.909,428.754,171.218,29.776,155.573
C00604=1056.665,7.159,428.739,171.219,29.778,155.573
C00605=1056.671,7.409,428.724,171.221,29.781,155.574
C00606=1056.676,7.658,428.709,171.223,29.783,155.574
C00607=1056.683,7.907,428.693,171.224,29.786,155.574
C00608=1056.690,8.156,428.678,171.226,29.788,155.575
C00609=1056.696,8.406,428.664,171.227,29.790,155.575
C00610=1056.702,8.656,428.649,171.229,29.792,155.575
C00611=1056.708,8.905,428.634,171.230,29.794,155.576
C00612=1056.714,9.154,428.619,171.232,29.796,155.576
C00613=1056.721,9.404,428.604,171.234,29.798,155.576
C00614=1056.727,9.654,428.589,171.236,29.801,155.576
C00615=1056.732,9.903,428.574,171.236,29.803,155.577
C00616=1056.739,10.153,428.559,171.238,29.805,155.577
C00617=1056.745,10.402,428.543,171.240,29.807,155.577
C00618=1056.752,10.651,428.528,171.242,29.810,155.578
C00619=1056.758,10.901,428.513,171.243,29.812,155.578
C00620=1056.764,11.151,428.499,171.244,29.814,155.578
C00621=1056.770,11.400,428.484,171.246,29.816,155.578
C00622=1056.777,11.649,428.469,171.248,29.819,155.579
C00623=1056.783,11.899,428.453,171.249,29.821,155.579
C00624=1056.789,12.148,428.438,171.251,29.823,155.579
C00625=1056.795,12.398,428.423,171.253,29.825,155.580
C00626=1056.802,12.648,428.408,171.254,29.827,155.580
C00627=1056.808,12.897,428.393,171.256,29.829,155.580
C00628=1056.814,13.146,428.378,171.257,29.832,155.581
C00629=1056.821,13.430,428.360,171.259,29.834,155.581
C00630=1056.828,13.715,428.343,171.261,29.836,155.581
C00631=1056.835,13.997,428.326,171.262,29.839,155.582
C00632=1056.842,14.282,428.309,171.264,29.842,155.582
C00633=1056.849,14.532,428.294,171.266,29.844,155.582
C00634=1056.855,14.781,428.277,171.268,29.846,155.583
C00635=1056.861,15.030,428.263,171.269,29.849,155.583
C00636=1056.867,15.280,428.248,171.270,29.851,155.583
C00637=1056.873,15.529,428.232,171.272,29.853,155.584
C00638=1056.879,15.779,428.217,171.274,29.855,155.584
C00639=1056.886,16.028,428.202,171.276,29.858,155.584
C00640=1056.892,16.278,428.186,171.277,29.860,155.585
C00641=1056.897,16.527,428.171,171.278,29.862,155.585
C00642=1056.903,16.776,428.155,171.280,29.864,155.585
C00643=1056.910,17.026,428.140,171.281,29.867,155.585
C00644=1056.916,17.275,428.125,171.283,29.869,155.586
C00645=1056.922,17.525,428.109,171.284,29.871,155.586
C00646=1056.928,17.774,428.094,171.286,29.874,155.586
C00647=1056.935,18.024,428.079,171.288,29.876,155.587
C00648=1056.941,18.273,428.062,171.289,29.878,155.587
C00649=1056.947,18.522,428.048,171.291,29.881,155.587
C00650=1056.952,18.771,428.032,171.292,29.883,155.588
C00651=1056.959,19.021,428.017,171.294,29.885,155.588
C00652=1056.965,19.271,428.002,171.295,29.888,155.588
C00653=1056.971,19.520,427.985,171.297,29.890,155.589
C00654=1056.978,19.770,427.970,171.299,29.892,155.589
C00655=1056.984,20.019,427.954,171.300,29.894,155.589
C00656=1056.990,20.269,427.939,171.301,29.897,155.590
C00657=1056.996,20.518,427.923,171.303,29.899,155.590
C00658=1057.002,20.768,427.908,171.305,29.902,155.590
C00659=1057.008,21.017,427.892,171.307,29.904,155.591
C00660=1057.014,21.266,427.877,171.307,29.906,155.591
C00661=1057.020,21.515,427.861,171.309,29.908,155.591
C00662=1057.026,21.765,427.846,171.311,29.911,155.591
C00663=1057.032,22.014,427.830,171.313,29.913,155.592
C00664=1057.039,22.264,427.815,171.313,29.915,155.592
C00665=1057.045,22.513,427.799,171.315,29.917,155.592
C00666=1057.051,22.763,427.784,171.317,29.920,155.593
C00667=1057.057,23.012,427.767,171.319,29.922,155.593
C00668=1057.063,23.262,427.752,171.321,29.925,155.593
C00669=1057.069,23.511,427.736,171.321,29.927,155.594
C00670=1057.076,23.761,427.721,171.323,29.929,155.594
C00671=1057.082,24.011,427.705,171.325,29.931,155.594
C00672=1057.088,24.260,427.689,171.327,29.934,155.595
C00673=1057.094,24.510,427.674,171.327,29.936,155.595
C00674=1057.100,24.759,427.658,171.329,29.938,155.595
C00675=1057.107,25.008,427.642,171.331,29.940,155.596
C00676=1057.112,25.258,427.626,171.333,29.943,155.596
C00677=1057.119,25.507,427.611,171.333,29.945,155.596
C00678=1057.125,25.756,427.594,171.335,29.947,155.597
C00679=1057.131,26.006,427.579,171.337,29.950,155.597
C00680=1057.137,26.255,427.563,171.339,29.952,155.597
C00681=1057.143,26.505,427.547,171.340,29.954,155.598
C00682=1057.150,26.754,427.532,171.341,29.957,155.598
C00683=1057.155,27.004,427.516,171.343,29.959,155.598
C00684=1057.162,27.253,427.500,171.345,29.961,155.599
C00685=1057.168,27.503,427.485,171.346,29.964,155.599
C00686=1057.174,27.752,427.468,171.347,29.966,155.599
C00687=1057.180,28.001,427.453,171.349,29.969,155.600
C00688=1057.186,28.251,427.437,171.351,29.971,155.600
C00689=1057.192,28.500,427.421,171.353,29.973,155.600
C00690=1057.199,28.749,427.405,171.354,29.976,155.601
C00691=1057.205,28.999,427.389,171.355,29.978,155.601
C00692=1057.210,29.249,427.373,171.357,29.981,155.601
C00693=1057.217,29.534,427.354,171.359,29.983,155.602
C00694=1057.224,29.818,427.337,171.360,29.985,155.602
C00695=1057.231,30.104,427.319,171.362,29.988,155.602
C00696=1057.238,30.389,427.301,171.364,29.991,155.603
C00697=1057.244,30.638,427.284,171.365,29.994,155.603
C00698=1057.251,30.888,427.269,171.367,29.996,155.603
C00699=1057.257,31.137,427.252,171.368,29.998,155.604
C00700=1057.263,31.386,427.236,171.370,30.001,155.604
C00701=1057.268,31.636,427.220,171.372,30.003,155.604
C00702=1057.274,31.886,427.204,171.373,30.005,155.605
C00703=1057.281,32.135,427.189,171.374,30.007,155.605
C00704=1057.287,32.385,427.172,171.376,30.010,155.606
C00705=1057.293,32.634,427.156,171.378,30.012,155.606
C00706=1057.299,32.883,427.139,171.379,30.015,155.606
C00707=1057.306,33.132,427.124,171.380,30.017,155.607
C00708=1057.312,33.382,427.108,171.382,30.019,155.607
C00709=1057.318,33.631,427.091,171.384,30.022,155.607
C00710=1057.323,33.881,427.076,171.385,30.024,155.608
C00711=1057.329,34.130,427.060,171.386,30.027,155.608
C00712=1057.336,34.379,427.044,171.388,30.029,155.608
C00713=1057.342,34.629,427.028,171.390,30.032,155.609
C00714=1057.348,34.878,427.011,171.391,30.034,155.609
C00715=1057.355,35.128,426.995,171.393,30.036,155.609
C00716=1057.361,35.378,426.978,171.394,30.038,155.610
C00717=1057.366,35.627,426.962,171.396,30.041,155.610
C00718=1057.373,35.876,426.947,171.397,30.043,155.610
C00719=1057.379,36.125,426.930,171.399,30.045,155.611
C00720=1057.385,36.375,426.914,171.400,30.048,155.611
C00721=1057.391,36.624,426.898,171.402,30.050,155.611
C00722=1057.397,36.873,426.882,171.404,30.052,155.612
C00723=1057.404,37.123,426.865,171.405,30.055,155.612
C00724=1057.410,37.372,426.849,171.406,30.057,155.612
C00725=1057.416,37.622,426.833,171.408,30.060,155.613
C00726=1057.422,37.871,426.817,171.410,30.062,155.613
C00727=1057.428,38.120,426.800,171.411,30.065,155.613
C00728=1057.434,38.370,426.784,171.412,30.067,155.614
C00729=1057.440,38.619,426.768,171.414,30.069,155.614
C00730=1057.447,38.869,426.751,171.416,30.072,155.614
C00731=1057.452,39.119,426.735,171.417,30.074,155.615
C00732=1057.459,39.367,426.718,171.418,30.076,155.615
C00733=1057.465,39.617,426.702,171.420,30.079,155.615
C00734=1057.471,39.866,426.686,171.422,30.081,155.616
C00735=1057.477,40.115,426.669,171.423,30.084,155.616
C00736=1057.483,40.365,426.653,171.424,30.086,155.616
C00737=1057.489,40.615,426.636,171.426,30.089,155.617
C00738=1057.495,40.864,426.620,171.428,30.091,155.617
C00739=1057.501,41.113,426.604,171.430,30.093,155.617
C00740=1057.507,41.362,426.587,171.430,30.096,155.618
C00741=1057.513,41.611,426.571,171.432,30.098,155.618
C00742=1057.519,41.861,426.554,171.434,30.101,155.619
C00743=1057.526,42.111,426.538,171.436,30.103,155.619
C00744=1057.532,42.360,426.522,171.436,30.106,155.619
C00745=1057.537,42.609,426.504,171.438,30.108,155.620
C00746=1057.543,42.859,426.488,171.440,30.111,155.620
C00747=1057.549,43.108,426.471,171.441,30.112,155.620
C00748=1057.556,43.358,426.455,171.442,30.115,155.621
C00749=1057.562,43.607,426.439,171.444,30.117,155.621
C00750=1057.568,43.856,426.422,171.446,30.120,155.621
C00751=1057.574,44.105,426.405,171.447,30.122,155.622
C00752=1057.579,44.355,426.389,171.449,30.125,155.622
C00753=1057.586,44.605,426.372,171.450,30.128,155.622
C00754=1057.592,44.854,426.355,171.452,30.130,155.623
C00755=1057.598,45.103,426.339,171.453,30.132,155.623
C00756=1057.603,45.353,426.322,171.455,30.135,155.624
C00757=1057.610,45.638,426.303,171.456,30.138,155.624
C00758=1057.617,45.923,426.284,171.458,30.140,155.624
C00759=1057.624,46.208,426.264,171.460,30.143,155.625
C00760=1057.631,46.493,426.245,171.461,30.146,155.625
C00761=1057.637,46.743,426.229,171.463,30.149,155.626
C00762=1057.642,46.993,426.212,171.464,30.151,155.626
C00763=1057.649,47.241,426.195,171.466,30.153,155.626
C00764=1057.655,47.491,426.179,171.468,30.156,155.627
C00765=1057.660,47.741,426.161,171.469,30.158,155.627
C00766=1057.667,47.990,426.144,171.470,30.161,155.627
C00767=1057.673,48.239,426.128,171.472,30.164,155.628
C00768=1057.679,48.488,426.111,171.474,30.166,155.628
C00769=1057.684,48.737,426.094,171.475,30.168,155.628
C00770=1057.691,48.987,426.077,171.476,30.171,155.629
C00771=1057.697,49.236,426.061,171.478,30.173,155.629
C00772=1057.702,49.486,426.044,171.480,30.176,155.630
C00773=1057.709,49.735,426.027,171.481,30.178,155.630
C00774=1057.715,49.985,426.010,171.482,30.181,155.630
C00775=1057.720,50.234,425.993,171.484,30.183,155.631
C00776=1057.726,50.483,425.976,171.486,30.185,155.631
C00777=1057.733,50.732,425.959,171.487,30.188,155.631
C00778=1057.739,50.982,425.943,171.488,30.190,155.632
C00779=1057.745,51.231,425.925,171.490,30.193,155.632
C00780=1057.751,51.481,425.909,171.492,30.196,155.632
C00781=1057.758,51.730,425.892,171.493,30.198,155.633
C00782=1057.763,51.979,425.875,171.494,30.200,155.633
C00783=1057.769,52.228,425.858,171.496,30.202,155.633
C00784=1057.776,52.478,425.841,171.498,30.205,155.634
C00785=1057.781,52.727,425.824,171.499,30.208,155.634
C00786=1057.787,52.976,425.807,171.500,30.210,155.635
C00787=1057.794,53.226,425.790,171.502,30.213,155.635
C00788=1057.799,53.476,425.773,171.504,30.215,155.635
C00789=1057.805,53.724,425.756,171.505,30.217,155.636
C00790=1057.811,53.975,425.739,171.507,30.220,155.636
C00791=1057.817,54.223,425.722,171.508,30.222,155.636
C00792=1057.824,54.472,425.705,171.510,30.225,155.637
C00793=1057.830,54.722,425.688,171.511,30.227,155.637
C00794=1057.836,54.971,425.671,171.513,30.230,155.638
C00795=1057.842,55.221,425.654,171.514,30.232,155.638
C00796=1057.848,55.470,425.637,171.515,30.234,155.638
C00797=1057.854,55.719,425.620,171.517,30.237,155.639
C00798=1057.861,55.969,425.603,171.519,30.239,155.639
C00799=1057.866,56.218,425.586,171.520,30.242,155.639
C00800=1057.872,56.467,425.569,171.521,30.244,155.640
C00801=1057.879,56.717,425.552,171.523,30.246,155.640
C00802=1057.884,56.966,425.534,171.525,30.249,155.640
C00803=1057.891,57.215,425.517,171.527,30.251,155.641
C00804=1057.897,57.465,425.500,171.527,30.254,155.641
C00805=1057.903,57.714,425.483,171.529,30.256,155.641
C00806=1057.910,57.963,425.466,171.531,30.259,155.642
C00807=1057.915,58.213,425.449,171.533,30.261,155.642
C00808=1057.922,58.462,425.432,171.533,30.263,155.643
C00809=1057.927,58.711,425.414,171.535,30.266,155.643
C00810=1057.934,58.961,425.398,171.537,30.268,155.643
C00811=1057.940,59.210,425.381,171.539,30.271,155.644
C00812=1057.946,59.460,425.363,171.540,30.273,155.644
C00813=1057.952,59.709,425.346,171.541,30.276,155.644
C00814=1057.958,59.959,425.328,171.543,30.278,155.645
C00815=1057.965,60.208,425.311,171.544,30.280,155.645
C00816=1057.971,60.456,425.294,171.546,30.283,155.645
C00817=1057.977,60.706,425.277,171.547,30.285,155.646
C00818=1057.983,60.955,425.260,171.549,30.288,155.646
C00819=1057.989,61.205,425.242,171.550,30.290,155.646
C00820=1057.995,61.454,425.225,171.552,30.293,155.647
C00821=1058.003,61.739,425.205,171.554,30.295,155.647
C00822=1058.010,62.024,425.186,171.555,30.298,155.648
C00823=1058.017,62.308,425.166,171.557,30.301,155.648
C00824=1058.023,62.594,425.146,171.559,30.304,155.648
C00825=1058.030,62.843,425.129,171.561,30.306,155.649
C00826=1058.036,63.092,425.112,171.562,30.308,155.649
C00827=1058.043,63.342,425.094,171.563,30.311,155.650
C00828=1058.049,63.591,425.076,171.565,30.313,155.650
C00829=1058.055,63.840,425.059,171.567,30.316,155.650
C00830=1058.062,64.090,425.043,171.568,30.318,155.651
C00831=1058.067,64.339,425.025,171.569,30.320,155.651
C00832=1058.073,64.589,425.007,171.571,30.323,155.651
C00833=1058.079,64.838,424.990,171.573,30.325,155.652
C00834=1058.086,65.087,424.972,171.575,30.328,155.652
C00835=1058.091,65.336,424.955,171.575,30.331,155.652
C00836=1058.098,65.586,424.937,171.577,30.333,155.653
C00837=1058.103,65.835,424.920,171.579,30.335,155.653
C00838=1058.110,66.085,424.902,171.581,30.338,155.654
C00839=1058.116,66.333,424.885,171.581,30.340,155.654
C00840=1058.122,66.583,424.867,171.583,30.343,155.654
C00841=1058.127,66.832,424.849,171.585,30.346,155.655
C00842=1058.134,67.081,424.832,171.586,30.347,155.655
C00843=1058.140,67.331,424.814,171.588,30.350,155.655
C00844=1058.146,67.580,424.797,171.589,30.353,155.656
C00845=1058.152,67.829,424.780,171.591,30.355,155.656
C00846=1058.158,68.079,424.762,171.592,30.358,155.657
C00847=1058.164,68.328,424.744,171.594,30.360,155.657
C00848=1058.170,68.578,424.726,171.596,30.362,155.657
C00849=1058.176,68.826,424.709,171.597,30.365,155.658
C00850=1058.182,69.076,424.691,171.598,30.368,155.658
C00851=1058.188,69.325,424.674,171.600,30.370,155.658
C00852=1058.194,69.575,424.656,171.602,30.373,155.659
C00853=1058.201,69.824,424.638,171.603,30.375,155.659
C00854=1058.206,70.073,424.621,171.604,30.377,155.659
C00855=1058.213,70.322,424.602,171.606,30.380,155.660
C00856=1058.218,70.571,424.585,171.608,30.383,155.660
C00857=1058.224,70.821,424.567,171.609,30.385,155.661
C00858=1058.230,71.070,424.549,171.610,30.387,155.661
C00859=1058.237,71.320,424.532,171.612,30.390,155.661
C00860=1058.242,71.569,424.514,171.614,30.393,155.662
C00861=1058.248,71.818,424.496,171.615,30.395,155.662
C00862=1058.255,72.068,424.478,171.616,30.397,155.662
C00863=1058.260,72.317,424.460,171.618,30.400,155.663
C00864=1058.267,72.566,424.442,171.620,30.403,155.663
C00865=1058.272,72.815,424.425,171.621,30.405,155.664
C00866=1058.279,73.065,424.407,171.623,30.407,155.664
C00867=1058.285,73.313,424.389,171.624,30.410,155.664
C00868=1058.291,73.563,424.371,171.626,30.412,155.665
C00869=1058.297,73.813,424.353,171.627,30.415,155.665
C00870=1058.302,74.062,424.335,171.629,30.418,155.666
C00871=1058.309,74.311,424.317,171.630,30.420,155.666
C00872=1058.315,74.561,424.299,171.631,30.422,155.666
C00873=1058.321,74.810,424.281,171.633,30.425,155.667
C00874=1058.327,75.059,424.263,171.635,30.428,155.667
C00875=1058.333,75.307,424.246,171.637,30.430,155.667
C00876=1058.339,75.557,424.228,171.637,30.432,155.668
C00877=1058.345,75.807,424.210,171.639,30.435,155.668
C00878=1058.351,76.056,424.192,171.641,30.438,155.669
C00879=1058.357,76.305,424.174,171.643,30.440,155.669
C00880=1058.364,76.555,424.156,171.644,30.442,155.669
C00881=1058.369,76.804,424.138,171.645,30.445,155.670
C00882=1058.375,77.053,424.119,171.647,30.447,155.670
C00883=1058.382,77.303,424.102,171.649,30.450,155.670
C00884=1058.387,77.552,424.084,171.650,30.452,155.671
C00885=1058.395,77.836,424.063,171.651,30.455,155.671
C00886=1058.401,78.121,424.042,171.653,30.458,155.672
C00887=1058.408,78.406,424.022,171.655,30.461,155.672
C00888=1058.415,78.691,424.001,171.657,30.464,155.673
C00889=1058.421,78.939,423.983,171.658,30.467,155.673
C00890=1058.427,79.189,423.965,171.660,30.469,155.673
C00891=1058.433,79.439,423.947,171.661,30.471,155.674
C00892=1058.438,79.688,423.928,171.663,30.474,155.674
C00893=1058.445,79.937,423.910,171.665,30.477,155.675
C00894=1058.451,80.186,423.892,171.666,30.479,155.675
C00895=1058.457,80.435,423.874,171.667,30.481,155.675
C00896=1058.463,80.685,423.856,171.669,30.484,155.676
C00897=1058.469,80.934,423.838,171.671,30.487,155.676
C00898=1058.474,81.183,423.819,171.672,30.489,155.676
C00899=1058.480,81.433,423.801,171.673,30.492,155.677
C00900=1058.487,81.682,423.782,171.675,30.494,155.677
C00901=1058.492,81.931,423.765,171.677,30.497,155.678
C00902=1058.499,82.180,423.746,171.679,30.499,155.678
C00903=1058.505,82.430,423.728,171.679,30.502,155.678
C00904=1058.510,82.679,423.709,171.681,30.504,155.679
C00905=1058.516,82.928,423.691,171.683,30.507,155.679
C00906=1058.522,83.177,423.673,171.685,30.510,155.679
C00907=1058.529,83.427,423.655,171.686,30.512,155.680
C00908=1058.534,83.676,423.636,171.687,30.515,155.680
C00909=1058.540,83.926,423.618,171.689,30.517,155.681
C00910=1058.546,84.175,423.599,171.691,30.520,155.681
C00911=1058.552,84.423,423.581,171.692,30.522,155.681
C00912=1058.558,84.673,423.563,171.694,30.525,155.682
C00913=1058.565,84.922,423.544,171.695,30.527,155.682
C00914=1058.571,85.172,423.526,171.697,30.530,155.683
C00915=1058.576,85.421,423.507,171.698,30.532,155.683
C00916=1058.582,85.670,423.489,171.700,30.535,155.683
C00917=1058.588,85.919,423.471,171.702,30.537,155.684
C00918=1058.595,86.169,423.452,171.703,30.540,155.684
C00919=1058.601,86.418,423.434,171.704,30.542,155.685
C00920=1058.606,86.667,423.415,171.706,30.545,155.685
C00921=1058.612,86.916,423.397,171.708,30.547,155.685
C00922=1058.619,87.165,423.378,171.709,30.550,155.686
C00923=1058.625,87.415,423.360,171.710,30.552,155.686
C00924=1058.631,87.663,423.342,171.712,30.555,155.686
C00925=1058.636,87.913,423.323,171.714,30.557,155.687
C00926=1058.643,88.163,423.305,171.716,30.560,155.687
C00927=1058.649,88.412,423.286,171.716,30.562,155.688
C00928=1058.655,88.661,423.267,171.718,30.564,155.688
C00929=1058.661,88.911,423.249,171.720,30.567,155.688
C00930=1058.667,89.159,423.231,171.722,30.570,155.689
C00931=1058.673,89.408,423.212,171.723,30.572,155.689
C00932=1058.679,89.658,423.193,171.724,30.574,155.689
C00933=1058.685,89.908,423.175,171.726,30.577,155.690
C00934=1058.691,90.157,423.156,171.728,30.580,155.690
C00935=1058.698,90.406,423.137,171.729,30.582,155.691
C00936=1058.703,90.654,423.119,171.731,30.584,155.691
C00937=1058.709,90.904,423.100,171.732,30.587,155.691
C00938=1058.715,91.153,423.082,171.734,30.590,155.692
C00939=1058.721,91.403,423.063,171.735,30.592,155.692
C00940=1058.727,91.652,423.044,171.737,30.595,155.693
C00941=1058.733,91.901,423.025,171.739,30.598,155.693
C00942=1058.739,92.150,423.007,171.740,30.600,155.693
C00943=1058.745,92.399,422.988,171.741,30.602,155.694
C00944=1058.751,92.649,422.969,171.743,30.605,155.694
C00945=1058.760,93.045,422.939,171.746,30.609,155.695
C00946=1058.770,93.442,422.910,171.748,30.613,155.695
C00947=1058.779,93.840,422.879,171.751,30.617,155.696
C00948=1058.788,94.237,422.849,171.753,30.621,155.697
C00949=1058.795,94.511,422.829,171.754,30.624,155.697
C00950=1058.802,94.785,422.808,171.756,30.627,155.698
C00951=1058.808,95.034,422.789,171.758,30.630,155.698
C00952=1058.813,95.283,422.770,171.760,30.632,155.698
C00953=1058.819,95.532,422.752,171.762,30.635,155.699
C00954=1058.825,95.781,422.732,171.762,30.637,155.699
C00955=1058.832,96.030,422.714,171.764,30.640,155.699
C00956=1058.837,96.280,422.694,171.766,30.643,155.700
C00957=1058.844,96.529,422.676,171.768,30.645,155.700
C00958=1058.849,96.778,422.657,171.769,30.647,155.701
C00959=1058.856,97.028,422.638,171.770,30.650,155.701
C00960=1058.862,97.277,422.619,171.772,30.653,155.701
C00961=1058.868,97.526,422.600,171.774,30.655,155.702
C00962=1058.873,97.775,422.581,171.775,30.658,155.702
C00963=1058.879,98.024,422.563,171.777,30.660,155.703
C00964=1058.885,98.273,422.543,171.778,30.663,155.703
C00965=1058.892,98.523,422.525,171.780,30.665,155.703
C00966=1058.897,98.772,422.505,171.782,30.668,155.704
C00967=1058.904,99.021,422.487,171.783,30.670,155.704
C00968=1058.909,99.271,422.468,171.785,30.673,155.705
C00969=1058.916,99.519,422.448,171.786,30.675,155.705
C00970=1058.922,99.768,422.429,171.788,30.678,155.705
C00971=1058.928,100.018,422.410,171.789,30.680,155.706
C00972=1058.934,100.267,422.391,171.791,30.683,155.706
C00973=1058.940,100.516,422.372,171.793,30.685,155.706
C00974=1058.946,100.766,422.353,171.794,30.688,155.707
C00975=1058.952,101.015,422.334,171.796,30.691,155.707
C00976=1058.958,101.264,422.315,171.797,30.693,155.708
C00977=1058.964,101.513,422.295,171.799,30.695,155.708
C00978=1058.970,101.762,422.276,171.801,30.698,155.708
C00979=1058.976,102.012,422.257,171.802,30.701,155.709
C00980=1058.982,102.261,422.238,171.803,30.703,155.709
C00981=1058.988,102.510,422.219,171.805,30.706,155.710
C00982=1058.993,102.758,422.199,171.807,30.709,155.710
C00983=1058.999,103.008,422.180,171.808,30.711,155.710
C00984=1059.005,103.257,422.161,171.810,30.714,155.711
C00985=1059.011,103.506,422.142,171.811,30.716,155.711
C00986=1059.017,103.755,422.122,171.813,30.719,155.712
C00987=1059.023,104.005,422.103,171.815,30.721,155.712
C00988=1059.028,104.254,422.084,171.816,30.724,155.712
C00989=1059.035,104.503,422.065,171.817,30.726,155.713
C00990=1059.041,104.752,422.045,171.819,30.729,155.713
C00991=1059.046,105.002,422.026,171.821,30.732,155.714
C00992=1059.052,105.251,422.007,171.823,30.734,155.714
C00993=1059.059,105.499,421.987,171.824,30.737,155.715
C00994=1059.064,105.749,421.968,171.825,30.739,155.715
C00995=1059.070,105.998,421.949,171.827,30.742,155.715
C00996=1059.076,106.247,421.929,171.829,30.744,155.716
C00997=1059.082,106.497,421.910,171.831,30.747,155.716
C00998=1059.088,106.746,421.891,171.832,30.750,155.716
C00999=1059.094,106.995,421.871,171.833,30.752,155.717
C01000=1059.100,107.244,421.852,171.835,30.755,155.717
C01001=1059.106,107.493,421.832,171.837,30.757,155.718
C01002=1059.112,107.743,421.812,171.839,30.760,155.718
C01003=1059.118,107.992,421.793,171.841,30.762,155.718
C01004=1059.124,108.241,421.774,171.841,30.765,155.719
C01005=1059.130,108.490,421.754,171.843,30.768,155.719
C01006=1059.136,108.740,421.735,171.845,30.770,155.720
C01007=1059.142,108.989,421.715,171.847,30.772,155.720
C01008=1059.148,109.238,421.696,171.849,30.775,155.720
C01009=1059.154,109.486,421.676,171.849,30.778,155.721
C01010=1059.160,109.736,421.657,171.851,30.780,155.721
C01011=1059.167,110.021,421.635,171.853,30.783,155.722
C01012=1059.174,110.305,421.613,171.855,30.786,155.722
C01013=1059.180,110.591,421.590,171.857,30.789,155.723
C01014=1059.187,110.875,421.567,171.858,30.792,155.723
C01015=1059.194,111.124,421.549,171.860,30.794,155.723
C01016=1059.200,111.373,421.529,171.862,30.797,155.724
C01017=1059.205,111.622,421.509,171.864,30.800,155.724
C01018=1059.211,111.871,421.489,171.866,30.802,155.725
C01019=1059.217,112.121,421.470,171.866,30.805,155.725
C01020=1059.224,112.370,421.450,171.868,30.808,155.725
C01021=1059.229,112.619,421.431,171.870,30.810,155.726
C01022=1059.235,112.868,421.411,171.872,30.812,155.726
C01023=1059.241,113.118,421.391,171.874,30.815,155.727
C01024=1059.247,113.367,421.372,171.875,30.818,155.727
C01025=1059.253,113.615,421.352,171.876,30.820,155.727
C01026=1059.259,113.865,421.332,171.878,30.823,155.728
C01027=1059.265,114.114,421.312,171.880,30.826,155.728
C01028=1059.270,114.363,421.293,171.882,30.828,155.729
C01029=1059.276,114.613,421.272,171.883,30.831,155.729
C01030=1059.282,114.862,421.252,171.884,30.833,155.730
C01031=1059.288,115.111,421.233,171.886,30.836,155.730
C01032=1059.294,115.360,421.213,171.888,30.839,155.730
C01033=1059.300,115.609,421.193,171.890,30.841,155.731
C01034=1059.305,115.858,421.173,171.891,30.844,155.731
C01035=1059.311,116.107,421.153,171.892,30.847,155.732
C01036=1059.317,116.356,421.133,171.894,30.849,155.732
C01037=1059.323,116.605,421.113,171.896,30.852,155.732
C01038=1059.329,116.854,421.094,171.898,30.855,155.733
C01039=1059.334,117.104,421.073,171.899,30.857,155.733
C01040=1059.340,117.353,421.053,171.901,30.860,155.734
C01041=1059.346,117.602,421.033,171.902,30.863,155.734
C01042=1059.352,117.851,421.014,171.904,30.865,155.734
C01043=1059.357,118.100,420.993,171.906,30.867,155.735
C01044=1059.363,118.349,420.974,171.908,30.870,155.735
C01045=1059.369,118.598,420.954,171.909,30.873,155.736
C01046=1059.376,118.848,420.934,171.910,30.875,155.736
C01047=1059.381,119.097,420.913,171.912,30.878,155.736
C01048=1059.387,119.346,420.893,171.914,30.880,155.737
C01049=1059.393,119.595,420.873,171.916,30.883,155.737
C01050=1059.399,119.844,420.854,171.917,30.886,155.738
C01051=1059.404,120.093,420.834,171.919,30.888,155.738
C01052=1059.410,120.343,420.813,171.920,30.891,155.739
C01053=1059.416,120.592,420.793,171.922,30.894,155.739
C01054=1059.422,120.841,420.773,171.924,30.896,155.739
C01055=1059.428,121.090,420.753,171.925,30.899,155.740
C01056=1059.434,121.338,420.733,171.927,30.902,155.740
C01057=1059.440,121.588,420.713,171.929,30.904,155.741
C01058=1059.446,121.837,420.693,171.930,30.907,155.741
C01059=1059.451,122.087,420.673,171.932,30.910,155.741
C01060=1059.457,122.335,420.653,171.933,30.912,155.742
C01061=1059.464,122.585,420.633,171.935,30.915,155.742
C01062=1059.470,122.834,420.613,171.937,30.917,155.743
C01063=1059.475,123.083,420.592,171.939,30.920,155.743
C01064=1059.481,123.332,420.572,171.941,30.922,155.743
C01065=1059.488,123.581,420.552,171.942,30.925,155.744
C01066=1059.493,123.830,420.531,171.943,30.927,155.744
C01067=1059.499,124.079,420.511,171.945,30.930,155.745
C01068=1059.505,124.328,420.491,171.947,30.933,155.745
C01069=1059.511,124.577,420.471,171.949,30.935,155.745
C01070=1059.517,124.827,420.450,171.951,30.938,155.746
C01071=1059.523,125.075,420.430,171.952,30.941,155.746
C01072=1059.529,125.325,420.410,171.953,30.943,155.747
C01073=1059.535,125.574,420.390,171.955,30.946,155.747
C01074=1059.541,125.823,420.370,171.957,30.949,155.748
C01075=1059.548,126.107,420.347,171.959,30.951,155.748
C01076=1059.555,126.393,420.323,171.961,30.954,155.748
C01077=1059.561,126.677,420.300,171.963,30.957,155.749
C01078=1059.568,126.962,420.277,171.965,30.960,155.749
C01079=1059.574,127.211,420.257,171.967,30.963,155.750
C01080=1059.580,127.460,420.236,171.968,30.965,155.750
C01081=1059.586,127.709,420.216,171.970,30.968,155.751
C01082=1059.592,127.958,420.195,171.971,30.971,155.751
C01083=1059.598,128.207,420.175,171.973,30.973,155.751
C01084=1059.604,128.456,420.155,171.975,30.976,155.752
C01085=1059.610,128.705,420.134,171.977,30.979,155.752
C01086=1059.616,128.955,420.114,171.979,30.981,155.753
C01087=1059.622,129.203,420.094,171.980,30.983,155.753
C01088=1059.627,129.452,420.073,171.981,30.986,155.753
C01089=1059.634,129.702,420.053,171.983,30.988,155.754
C01090=1059.640,129.950,420.032,171.985,30.991,155.754
C01091=1059.646,130.200,420.012,171.987,30.994,155.755
C01092=1059.652,130.449,419.992,171.989,30.996,155.755
C01093=1059.658,130.698,419.972,171.990,30.999,155.755
C01094=1059.664,130.947,419.951,171.992,31.001,155.756
C01095=1059.670,131.196,419.930,171.994,31.004,155.756
C01096=1059.677,131.445,419.910,171.996,31.006,155.757
C01097=1059.682,131.694,419.889,171.998,31.009,155.757
C01098=1059.688,131.943,419.869,171.999,31.012,155.757
C01099=1059.694,132.192,419.848,172.000,31.014,155.758
C01100=1059.700,132.441,419.827,172.002,31.017,155.758
C01101=1059.706,132.691,419.807,172.004,31.020,155.759
C01102=1059.711,132.940,419.786,172.006,31.022,155.759
C01103=1059.718,133.188,419.765,172.008,31.025,155.759
C01104=1059.724,133.438,419.745,172.009,31.028,155.760
C01105=1059.729,133.687,419.724,172.011,31.030,155.760
C01106=1059.735,133.935,419.703,172.013,31.033,155.761
C01107=1059.741,134.185,419.682,172.014,31.035,155.761
C01108=1059.747,134.434,419.662,172.016,31.038,155.762
C01109=1059.753,134.683,419.641,172.018,31.041,155.762
C01110=1059.758,134.932,419.620,172.019,31.043,155.762
C01111=1059.764,135.181,419.600,172.021,31.046,155.763
C01112=1059.770,135.430,419.579,172.023,31.049,155.763
C01113=1059.776,135.679,419.558,172.025,31.051,155.764
C01114=1059.783,135.928,419.537,172.027,31.054,155.764
C01115=1059.788,136.178,419.516,172.028,31.057,155.764
C01116=1059.794,136.427,419.496,172.030,31.059,155.765
C01117=1059.800,136.676,419.475,172.031,31.062,155.765
C01118=1059.805,136.925,419.454,172.033,31.064,155.766
C01119=1059.811,137.174,419.433,172.035,31.067,155.766
C01120=1059.817,137.423,419.413,172.037,31.070,155.767
C01121=1059.824,137.672,419.391,172.038,31.072,155.767
C01122=1059.829,137.921,419.371,172.040,31.075,155.767
C01123=1059.836,138.170,419.350,172.042,31.078,155.768
C01124=1059.841,138.419,419.329,172.044,31.080,155.768
C01125=1059.847,138.668,419.307,172.046,31.083,155.769
C01126=1059.853,138.917,419.287,172.048,31.086,155.769
C01127=1059.859,139.166,419.266,172.049,31.088,155.770
C01128=1059.865,139.415,419.245,172.051,31.091,155.770
C01129=1059.871,139.665,419.224,172.053,31.094,155.770
C01130=1059.877,139.913,419.204,172.054,31.096,155.771
C01131=1059.883,140.163,419.182,172.056,31.099,155.771
C01132=1059.888,140.412,419.161,172.057,31.101,155.772
C01133=1059.894,140.661,419.140,172.059,31.104,155.772
C01134=1059.900,140.909,419.119,172.061,31.107,155.772
C01135=1059.906,141.159,419.098,172.063,31.109,155.773
C01136=1059.912,141.407,419.077,172.065,31.112,155.773
C01137=1059.918,141.657,419.055,172.067,31.115,155.774
C01138=1059.924,141.906,419.035,172.068,31.118,155.774
C01139=1059.930,142.190,419.011,172.070,31.121,155.775
C01140=1059.937,142.475,418.986,172.072,31.124,155.775
C01141=1059.944,142.759,418.962,172.075,31.127,155.776
C01142=1059.950,143.044,418.938,172.077,31.130,155.776
C01143=1059.956,143.293,418.917,172.078,31.133,155.777
C01144=1059.962,143.542,418.895,172.080,31.135,155.777
C01145=1059.968,143.791,418.875,172.082,31.138,155.777
C01146=1059.974,144.040,418.853,172.084,31.141,155.778
C01147=1059.979,144.289,418.832,172.085,31.143,155.778
C01148=1059.985,144.538,418.810,172.087,31.146,155.779
C01149=1059.991,144.787,418.790,172.088,31.148,155.779
C01150=1059.998,145.036,418.769,172.090,31.152,155.780
C01151=1060.003,145.285,418.747,172.092,31.154,155.780
C01152=1060.009,145.534,418.726,172.094,31.157,155.780
C01153=1060.015,145.784,418.705,172.096,31.159,155.781
C01154=1060.021,146.032,418.683,172.098,31.162,155.781
C01155=1060.027,146.281,418.662,172.099,31.165,155.782
C01156=1060.032,146.530,418.641,172.101,31.167,155.782
C01157=1060.039,146.779,418.619,172.103,31.170,155.782
C01158=1060.044,147.029,418.598,172.105,31.173,155.783
C01159=1060.050,147.277,418.577,172.107,31.175,155.783
C01160=1060.056,147.527,418.555,172.109,31.178,155.784
C01161=1060.062,147.775,418.534,172.110,31.181,155.784
C01162=1060.068,148.024,418.512,172.112,31.183,155.785
C01163=1060.074,148.274,418.491,172.114,31.186,155.785
C01164=1060.080,148.522,418.469,172.116,31.189,155.785
C01165=1060.085,148.772,418.448,172.118,31.191,155.786
C01166=1060.091,149.020,418.427,172.120,31.194,155.786
C01167=1060.097,149.270,418.405,172.121,31.197,155.787
C01168=1060.103,149.519,418.384,172.123,31.200,155.787
C01169=1060.109,149.767,418.363,172.125,31.202,155.788
C01170=1060.115,150.016,418.341,172.127,31.205,155.788
C01171=1060.121,150.265,418.320,172.129,31.208,155.788
C01172=1060.127,150.514,418.298,172.130,31.210,155.789
C01173=1060.133,150.763,418.276,172.132,31.213,155.789
C01174=1060.138,151.012,418.254,172.134,31.216,155.790
C01175=1060.144,151.261,418.233,172.136,31.219,155.790
C01176=1060.150,151.511,418.211,172.138,31.221,155.791
C01177=1060.156,151.759,418.190,172.140,31.224,155.791
C01178=1060.162,152.008,418.168,172.141,31.227,155.791
C01179=1060.168,152.258,418.147,172.143,31.229,155.792
C01180=1060.173,152.506,418.125,172.145,31.232,155.792
C01181=1060.179,152.756,418.103,172.147,31.235,155.793
C01182=1060.185,153.005,418.082,172.149,31.237,155.793
C01183=1060.191,153.253,418.060,172.151,31.241,155.794
C01184=1060.197,153.502,418.039,172.152,31.243,155.794
C01185=1060.203,153.752,418.017,172.154,31.246,155.795
C01186=1060.208,154.000,417.994,172.156,31.248,155.795
C01187=1060.214,154.249,417.973,172.158,31.251,155.795
C01188=1060.220,154.498,417.951,172.160,31.254,155.796
C01189=1060.226,154.747,417.930,172.162,31.256,155.796
C01190=1060.232,154.996,417.908,172.163,31.259,155.797
C01191=1060.238,155.246,417.886,172.165,31.262,155.797
C01192=1060.244,155.495,417.864,172.167,31.265,155.798
C01193=1060.250,155.743,417.842,172.169,31.267,155.798
C01194=1060.256,155.992,417.821,172.171,31.270,155.798
C01195=1060.261,156.241,417.799,172.173,31.273,155.799
C01196=1060.267,156.490,417.777,172.175,31.275,155.799
C01197=1060.273,156.739,417.756,172.176,31.279,155.800
C01198=1060.279,156.988,417.733,172.178,31.281,155.800
C01199=1060.285,157.237,417.711,172.180,31.284,155.801
C01200=1060.290,157.486,417.690,172.182,31.287,155.801
C01201=1060.296,157.735,417.668,172.184,31.289,155.801
C01202=1060.302,157.984,417.645,172.186,31.292,155.802
C01203=1060.308,158.268,417.621,172.187,31.295,155.802
C01204=1060.316,158.552,417.595,172.190,31.298,155.803
C01205=1060.322,158.837,417.571,172.192,31.302,155.803
C01206=1060.329,159.121,417.545,172.194,31.304,155.804
C01207=1060.335,159.370,417.524,172.196,31.307,155.804
C01208=1060.341,159.618,417.502,172.197,31.310,155.805
C01209=1060.346,159.868,417.479,172.199,31.313,155.805
C01210=1060.352,160.117,417.458,172.202,31.315,155.806
C01211=1060.359,160.365,417.435,172.204,31.318,155.806
C01212=1060.364,160.615,417.413,172.206,31.321,155.807
C01213=1060.370,160.863,417.392,172.208,31.324,155.807
C01214=1060.376,161.112,417.369,172.209,31.327,155.807
C01215=1060.382,161.362,417.347,172.211,31.329,155.808
C01216=1060.388,161.610,417.324,172.213,31.332,155.808
C01217=1060.392,161.859,417.302,172.215,31.335,155.809
C01218=1060.399,162.108,417.280,172.217,31.338,155.809
C01219=1060.404,162.357,417.258,172.219,31.341,155.810
C01220=1060.409,162.606,417.235,172.220,31.344,155.810
C01221=1060.416,162.855,417.214,172.222,31.346,155.811
C01222=1060.421,163.104,417.191,172.224,31.349,155.811
C01223=1060.427,163.353,417.169,172.226,31.352,155.812
C01224=1060.433,163.602,417.146,172.228,31.355,155.812
C01225=1060.438,163.851,417.124,172.230,31.358,155.813
C01226=1060.444,164.099,417.101,172.232,31.360,155.813
C01227=1060.450,164.349,417.080,172.233,31.364,155.814
C01228=1060.456,164.598,417.057,172.235,31.366,155.814
C01229=1060.460,164.846,417.035,172.237,31.369,155.814
C01230=1060.466,165.095,417.012,172.240,31.372,155.815
C01231=1060.472,165.345,416.990,172.242,31.375,155.815
C01232=1060.478,165.593,416.967,172.244,31.378,155.816
C01233=1060.484,165.842,416.944,172.245,31.381,155.816
C01234=1060.489,166.091,416.923,172.247,31.383,155.817
C01235=1060.495,166.340,416.900,172.249,31.386,155.817
C01236=1060.500,166.589,416.878,172.251,31.389,155.818
C01237=1060.506,166.838,416.855,172.253,31.392,155.818
C01238=1060.513,167.087,416.833,172.255,31.394,155.818
C01239=1060.518,167.336,416.810,172.256,31.398,155.819
C01240=1060.523,167.584,416.788,172.258,31.400,155.819
C01241=1060.529,167.833,416.765,172.260,31.404,155.820
C01242=1060.535,168.083,416.743,172.263,31.406,155.820
C01243=1060.541,168.331,416.720,172.265,31.409,155.821
C01244=1060.547,168.580,416.697,172.267,31.412,155.821
C01245=1060.552,168.829,416.674,172.268,31.415,155.822
C01246=1060.558,169.078,416.653,172.270,31.417,155.822
C01247=1060.564,169.327,416.630,172.272,31.421,155.823
C01248=1060.570,169.576,416.607,172.274,31.423,155.823
C01249=1060.575,169.824,416.584,172.276,31.426,155.824
C01250=1060.581,170.074,416.563,172.278,31.429,155.824
C01251=1060.587,170.323,416.540,172.280,31.432,155.825
C01252=1060.593,170.571,416.517,172.282,31.434,155.825
C01253=1060.598,170.820,416.494,172.284,31.438,155.825
C01254=1060.605,171.070,416.472,172.286,31.440,155.826
C01255=1060.610,171.318,416.449,172.288,31.443,155.826
C01256=1060.616,171.567,416.426,172.290,31.446,155.827
C01257=1060.622,171.816,416.403,172.292,31.449,155.827
C01258=1060.628,172.065,416.381,172.293,31.451,155.828
C01259=1060.634,172.314,416.358,172.295,31.455,155.828
C01260=1060.639,172.563,416.336,172.298,31.457,155.829
C01261=1060.645,172.812,416.313,172.300,31.460,155.829
C01262=1060.651,173.061,416.290,172.302,31.463,155.830
C01263=1060.657,173.310,416.268,172.304,31.466,155.830
C01264=1060.663,173.558,416.245,172.306,31.468,155.830
C01265=1060.669,173.807,416.222,172.307,31.472,155.831
C01266=1060.675,174.056,416.199,172.309,31.474,155.831
C01267=1060.681,174.340,416.173,172.312,31.478,155.832
C01268=1060.688,174.624,416.147,172.314,31.481,155.832
C01269=1060.695,174.907,416.121,172.317,31.484,155.833
C01270=1060.701,175.191,416.095,172.318,31.487,155.834
C01271=1060.707,175.440,416.072,172.320,31.490,155.834
C01272=1060.713,175.689,416.049,172.323,31.493,155.834
C01273=1060.719,175.938,416.027,172.325,31.496,155.835
C01274=1060.724,176.187,416.004,172.327,31.498,155.835
C01275=1060.730,176.436,415.981,172.329,31.502,155.836
C01276=1060.737,176.684,415.958,172.331,31.504,155.836
C01277=1060.742,176.933,415.935,172.332,31.507,155.837
C01278=1060.748,177.182,415.912,172.335,31.510,155.837
C01279=1060.754,177.432,415.889,172.337,31.513,155.838
C01280=1060.760,177.681,415.866,172.339,31.515,155.838
C01281=1060.766,177.930,415.843,172.341,31.519,155.839
C01282=1060.772,178.178,415.821,172.343,31.521,155.839
C01283=1060.778,178.427,415.797,172.345,31.524,155.839
C01284=1060.784,178.675,415.774,172.347,31.527,155.840
C01285=1060.790,178.924,415.751,172.349,31.530,155.840
C01286=1060.796,179.173,415.728,172.351,31.532,155.841
C01287=1060.801,179.422,415.705,172.353,31.536,155.841
C01288=1060.808,179.672,415.682,172.355,31.538,155.842
C01289=1060.813,179.921,415.659,172.358,31.542,155.842
C01290=1060.820,180.169,415.637,172.359,31.544,155.843
C01291=1060.826,180.417,415.613,172.361,31.547,155.843
C01292=1060.832,180.666,415.590,172.363,31.550,155.844
C01293=1060.837,180.915,415.567,172.365,31.553,155.844
C01294=1060.844,181.165,415.544,172.368,31.555,155.845
C01295=1060.849,181.414,415.521,172.370,31.559,155.845
C01296=1060.855,181.662,415.497,172.372,31.561,155.846
C01297=1060.861,181.911,415.474,172.373,31.564,155.846
C01298=1060.868,182.159,415.452,172.376,31.567,155.846
C01299=1060.874,182.409,415.429,172.378,31.570,155.847
C01300=1060.880,182.657,415.405,172.380,31.572,155.847
C01301=1060.886,182.906,415.382,172.382,31.575,155.848
C01302=1060.891,183.155,415.359,172.384,31.578,155.848
C01303=1060.897,183.404,415.336,172.387,31.581,155.849
C01304=1060.904,183.653,415.312,172.388,31.584,155.849
C01305=1060.910,183.902,415.289,172.390,31.587,155.850
C01306=1060.915,184.151,415.266,172.392,31.589,155.850
C01307=1060.921,184.399,415.243,172.395,31.593,155.851
C01308=1060.928,184.649,415.219,172.397,31.595,155.851
C01309=1060.934,184.897,415.196,172.399,31.598,155.852
C01310=1060.939,185.146,415.172,172.401,31.602,155.852
C01311=1060.944,185.395,415.149,172.403,31.604,155.853
C01312=1060.950,185.643,415.126,172.405,31.607,155.853
C01313=1060.955,185.893,415.102,172.407,31.611,155.854
C01314=1060.961,186.141,415.078,172.409,31.613,155.854
C01315=1060.967,186.391,415.054,172.411,31.616,155.855
C01316=1060.973,186.639,415.031,172.414,31.620,155.855
C01317=1060.979,186.888,415.008,172.416,31.622,155.856
C01318=1060.984,187.137,414.984,172.417,31.626,155.856
C01319=1060.990,187.385,414.961,172.419,31.628,155.856
C01320=1060.996,187.634,414.937,172.422,31.632,155.857
C01321=1061.002,187.884,414.913,172.424,31.635,155.858
C01322=1061.008,188.132,414.889,172.426,31.637,155.858
C01323=1061.013,188.381,414.866,172.428,31.640,155.859
C01324=1061.019,188.629,414.842,172.431,31.644,155.859
C01325=1061.024,188.878,414.818,172.432,31.646,155.859
C01326=1061.030,189.128,414.795,172.434,31.650,155.860
C01327=1061.036,189.376,414.771,172.436,31.653,155.861
C01328=1061.041,189.625,414.747,172.439,31.656,155.861
C01329=1061.047,189.873,414.724,172.441,31.659,155.862
C01330=1061.053,190.122,414.699,172.443,31.662,155.862
C01331=1061.060,190.406,414.673,172.445,31.665,155.863
C01332=1061.067,190.689,414.645,172.447,31.668,155.863
C01333=1061.072,190.973,414.619,172.450,31.672,155.864
C01334=1061.079,191.256,414.591,172.453,31.676,155.864
C01335=1061.085,191.504,414.567,172.455,31.679,155.865
C01336=1061.091,191.753,414.544,172.457,31.681,155.865
C01337=1061.097,192.003,414.520,172.459,31.685,155.866
C01338=1061.103,192.251,414.496,172.461,31.688,155.866
C01339=1061.108,192.500,414.473,172.463,31.690,155.867
C01340=1061.114,192.749,414.449,172.465,31.694,155.867
C01341=1061.120,192.998,414.424,172.468,31.697,155.868
C01342=1061.126,193.246,414.401,172.470,31.700,155.868
C01343=1061.132,193.495,414.376,172.472,31.703,155.869
C01344=1061.137,193.744,414.353,172.474,31.706,155.869
C01345=1061.143,193.993,414.329,172.476,31.709,155.870
C01346=1061.149,194.242,414.305,172.478,31.712,155.870
C01347=1061.155,194.490,414.281,172.480,31.715,155.871
C01348=1061.161,194.739,414.257,172.483,31.718,155.871
C01349=1061.167,194.988,414.234,172.485,31.721,155.872
C01350=1061.172,195.237,414.209,172.487,31.724,155.872
C01351=1061.178,195.485,414.186,172.490,31.727,155.873
C01352=1061.184,195.734,414.161,172.491,31.730,155.873
C01353=1061.190,195.983,414.137,172.493,31.733,155.874
C01354=1061.196,196.232,414.113,172.496,31.736,155.874
C01355=1061.202,196.480,414.089,172.498,31.739,155.875
C01356=1061.208,196.729,414.065,172.500,31.742,155.875
C01357=1061.214,196.978,414.041,172.503,31.746,155.876
C01358=1061.219,197.226,414.017,172.505,31.748,155.876
C01359=1061.226,197.476,413.993,172.507,31.751,155.877
C01360=1061.231,197.725,413.969,172.509,31.755,155.877
C01361=1061.238,197.973,413.945,172.511,31.757,155.878
C01362=1061.243,198.222,413.921,172.513,31.760,155.878
C01363=1061.249,198.470,413.897,172.516,31.764,155.879
C01364=1061.255,198.720,413.872,172.518,31.767,155.879
C01365=1061.261,198.968,413.849,172.520,31.769,155.880
C01366=1061.267,199.217,413.824,172.523,31.773,155.880
C01367=1061.272,199.466,413.800,172.524,31.776,155.881
C01368=1061.279,199.715,413.776,172.527,31.779,155.881
C01369=1061.284,199.963,413.751,172.529,31.782,155.882
C01370=1061.291,200.212,413.727,172.531,31.785,155.882
C01371=1061.296,200.460,413.703,172.534,31.788,155.883
C01372=1061.303,200.709,413.679,172.536,31.791,155.883
C01373=1061.308,200.958,413.654,172.538,31.794,155.884
C01374=1061.315,201.207,413.630,172.540,31.797,155.884
C01375=1061.320,201.455,413.606,172.542,31.800,155.885
C01376=1061.327,201.704,413.582,172.545,31.803,155.885
C01377=1061.332,201.953,413.558,172.547,31.806,155.886
C01378=1061.338,202.202,413.532,172.549,31.810,155.887
C01379=1061.344,202.450,413.508,172.552,31.813,155.887
C01380=1061.350,202.699,413.484,172.554,31.816,155.888
C01381=1061.356,202.948,413.460,172.557,31.819,155.888
C01382=1061.362,203.197,413.435,172.558,31.822,155.889
C01383=1061.367,203.445,413.410,172.560,31.825,155.889
C01384=1061.373,203.694,413.386,172.563,31.828,155.890
C01385=1061.378,203.943,413.361,172.565,31.831,155.890
C01386=1061.385,204.191,413.337,172.567,31.835,155.891
C01387=1061.391,204.440,413.312,172.570,31.838,155.891
C01388=1061.397,204.689,413.288,172.572,31.841,155.892
C01389=1061.402,204.938,413.264,172.574,31.844,155.892
C01390=1061.408,205.186,413.238,172.576,31.848,155.893
C01391=1061.414,205.436,413.214,172.578,31.851,155.893
C01392=1061.419,205.684,413.189,172.581,31.854,155.894
C01393=1061.426,205.933,413.165,172.583,31.857,155.895
C01394=1061.431,206.181,413.140,172.586,31.860,155.895
C01395=1061.456,207.230,413.036,172.761,31.944,155.903
C01396=1061.462,207.457,413.013,172.762,31.948,155.904
C01397=1061.467,207.685,412.990,172.764,31.951,155.905
C01398=1061.473,207.913,412.966,172.766,31.955,155.905
C01399=1061.479,208.140,412.943,172.768,31.959,155.906
C01400=1061.484,208.368,412.919,172.770,31.962,155.907
C01401=1061.490,208.595,412.896,172.772,31.966,155.907
C01402=1061.496,208.823,412.872,172.774,31.970,155.908
C01403=1061.501,209.051,412.849,172.775,31.973,155.909
C01404=1061.507,209.299,412.823,172.776,31.977,155.910
C01405=1061.514,209.548,412.798,172.779,31.982,155.910
C01406=1061.520,209.796,412.772,172.781,31.985,155.911
C01407=1061.525,210.045,412.746,172.783,31.989,155.912
C01408=1061.532,210.294,412.721,172.785,31.994,155.913
C01409=1061.538,210.542,412.695,172.787,31.997,155.913
C01410=1061.544,210.791,412.669,172.789,32.002,155.914
C01411=1061.550,211.040,412.644,172.791,32.005,155.915
C01412=1061.556,211.288,412.618,172.792,32.010,155.915
C01413=1061.562,211.536,412.592,172.794,32.013,155.916
C01414=1061.568,211.785,412.566,172.796,32.018,155.917
C01415=1061.574,212.034,412.541,172.798,32.021,155.918
C01416=1061.581,212.282,412.515,172.801,32.026,155.918
C01417=1061.586,212.531,412.489,172.803,32.030,155.919
C01418=1061.592,212.780,412.464,172.805,32.034,155.920
C01419=1061.599,213.028,412.438,172.807,32.038,155.921
C01420=1061.604,213.277,412.412,172.808,32.042,155.921
C01421=1061.610,213.526,412.386,172.810,32.046,155.922
C01422=1061.616,213.774,412.360,172.812,32.050,155.923
C01423=1061.622,214.023,412.334,172.814,32.054,155.924
C01424=1061.628,214.271,412.308,172.816,32.058,155.924
C01425=1061.634,214.520,412.282,172.819,32.062,155.925
C01426=1061.640,214.768,412.256,172.821,32.066,155.926
C01427=1061.646,215.017,412.230,172.823,32.070,155.927
C01428=1061.652,215.266,412.204,172.824,32.074,155.927
C01429=1061.659,215.514,412.178,172.826,32.078,155.928
C01430=1061.664,215.763,412.152,172.828,32.082,155.929
C01431=1061.671,216.011,412.126,172.830,32.086,155.929
C01432=1061.676,216.260,412.100,172.832,32.090,155.930
C01433=1061.683,216.508,412.074,172.835,32.094,155.931
C01434=1061.689,216.757,412.049,172.837,32.098,155.932
C01435=1061.695,217.005,412.022,172.839,32.102,155.932
C01436=1061.701,217.253,411.996,172.841,32.106,155.933
C01437=1061.708,217.503,411.970,172.842,32.110,155.934
C01438=1061.714,217.751,411.944,172.844,32.114,155.935
C01439=1061.720,218.000,411.918,172.846,32.118,155.935
C01440=1061.726,218.248,411.892,172.849,32.122,155.936
C01441=1061.732,218.497,411.865,172.851,32.126,155.937
C01442=1061.737,218.746,411.839,172.853,32.130,155.937
C01443=1061.744,218.994,411.813,172.855,32.134,155.938
C01444=1061.750,219.243,411.787,172.857,32.138,155.939
C01445=1061.756,219.491,411.761,172.859,32.142,155.940
C01446=1061.762,219.740,411.734,172.861,32.146,155.940
C01447=1061.768,219.988,411.709,172.863,32.150,155.941
C01448=1061.775,220.237,411.682,172.865,32.154,155.942
C01449=1061.781,220.486,411.656,172.867,32.158,155.943
C01450=1061.787,220.734,411.629,172.869,32.162,155.943
C01451=1061.793,220.983,411.604,172.871,32.166,155.944
C01452=1061.799,221.212,411.579,172.873,32.169,155.945
C01453=1061.804,221.442,411.555,172.875,32.173,155.945
C01454=1061.810,221.672,411.530,172.878,32.177,155.946
C01455=1061.816,221.903,411.505,172.880,32.180,155.947
C01456=1061.821,222.134,411.481,172.881,32.184,155.947
C01457=1061.827,222.364,411.456,172.883,32.188,155.948
C01458=1061.832,222.594,411.432,172.885,32.191,155.949
C01459=1061.838,222.823,411.407,172.887,32.195,155.949
C01460=1061.844,223.072,411.381,172.889,32.199,155.950
C01461=1061.850,223.320,411.355,172.891,32.203,155.951
C01462=1061.856,223.568,411.328,172.893,32.207,155.952
C01463=1061.862,223.817,411.301,172.895,32.211,155.952
C01464=1061.868,224.066,411.274,172.898,32.215,155.953
C01465=1061.874,224.314,411.249,172.900,32.219,155.954
C01466=1061.880,224.563,411.222,172.901,32.223,155.954
C01467=1061.886,224.812,411.195,172.903,32.227,155.955
C01468=1061.892,225.060,411.169,172.905,32.231,155.956
C01469=1061.898,225.308,411.142,172.908,32.235,155.957
C01470=1061.904,225.556,411.116,172.910,32.239,155.957
C01471=1061.911,225.806,411.089,172.912,32.243,155.958
C01472=1061.917,226.054,411.062,172.914,32.247,155.959
C01473=1061.922,226.302,411.036,172.916,32.250,155.960
C01474=1061.929,226.551,411.009,172.919,32.255,155.960
C01475=1061.935,226.799,410.983,172.921,32.259,155.961
C01476=1061.941,227.048,410.956,172.922,32.263,155.962
C01477=1061.947,227.297,410.929,172.924,32.266,155.963
C01478=1061.953,227.545,410.902,172.927,32.270,155.963
C01479=1061.959,227.794,410.876,172.929,32.274,155.964
C01480=1061.966,228.042,410.849,172.931,32.278,155.965
C01481=1061.972,228.291,410.823,172.933,32.282,155.965
C01482=1061.978,228.538,410.795,172.936,32.286,155.966
C01483=1061.984,228.787,410.768,172.938,32.290,155.967
C01484=1061.990,229.036,410.742,172.940,32.294,155.968
C01485=1061.996,229.285,410.715,172.942,32.298,155.968
C01486=1062.003,229.533,410.689,172.945,32.302,155.969
C01487=1062.009,229.781,410.662,172.946,32.306,155.970
C01488=1062.015,230.030,410.635,172.948,32.310,155.970
C01489=1062.021,230.278,410.608,172.950,32.314,155.971
C01490=1062.027,230.527,410.580,172.953,32.318,155.972
C01491=1062.033,230.776,410.553,172.955,32.321,155.973
C01492=1062.038,231.024,410.527,172.957,32.326,155.973
C01493=1062.045,231.273,410.500,172.959,32.329,155.974
C01494=1062.051,231.521,410.472,172.962,32.334,155.975
C01495=1062.057,231.769,410.446,172.964,32.337,155.976
C01496=1062.063,232.018,410.419,172.966,32.341,155.976
C01497=1062.069,232.266,410.391,172.968,32.345,155.977
C01498=1062.075,232.515,410.364,172.971,32.349,155.978
C01499=1062.081,232.764,410.338,172.972,32.353,155.978
C01500=1062.088,233.012,410.310,172.974,32.357,155.979
C01501=1062.094,233.260,410.283,172.977,32.361,155.980
C01502=1062.099,233.509,410.257,172.979,32.365,155.981
C01503=1062.106,233.757,410.229,172.981,32.369,155.981
C01504=1062.111,234.006,410.202,172.983,32.373,155.982
C01505=1062.118,234.255,410.175,172.986,32.377,155.983
C01506=1062.124,234.503,410.147,172.988,32.381,155.984
C01507=1062.129,234.751,410.121,172.990,32.385,155.984
C01508=1062.136,234.977,410.095,172.992,32.388,155.985
C01509=1062.141,235.203,410.071,172.994,32.392,155.986
C01510=1062.146,235.429,410.046,172.997,32.396,155.986
C01511=1062.152,235.655,410.021,172.999,32.399,155.987
C01512=1062.158,235.882,409.997,173.001,32.402,155.988
C01513=1062.163,236.107,409.972,173.002,32.406,155.988
C01514=1062.168,236.334,409.946,173.004,32.410,155.989
C01515=1062.174,236.560,409.921,173.006,32.413,155.990
C01516=1062.180,236.808,409.894,173.008,32.417,155.990
C01517=1062.186,237.057,409.867,173.011,32.421,155.991
C01518=1062.192,237.304,409.840,173.013,32.425,155.992
C01519=1062.198,237.554,409.813,173.015,32.429,155.992
C01520=1062.204,237.802,409.784,173.018,32.433,155.993
C01521=1062.210,238.051,409.758,173.020,32.437,155.994
C01522=1062.217,238.299,409.730,173.022,32.440,155.995
C01523=1062.223,238.547,409.703,173.025,32.444,155.995
C01524=1062.229,238.796,409.675,173.027,32.448,155.996
C01525=1062.235,239.044,409.648,173.029,32.452,155.997
C01526=1062.241,239.292,409.620,173.032,32.456,155.997
C01527=1062.247,239.541,409.593,173.033,32.460,155.998
C01528=1062.253,239.789,409.565,173.035,32.464,155.999
C01529=1062.260,240.038,409.537,173.038,32.468,156.000
C01530=1062.266,240.286,409.511,173.040,32.472,156.000
C01531=1062.271,240.535,409.482,173.042,32.475,156.001
C01532=1062.278,240.783,409.455,173.045,32.480,156.002
C01533=1062.284,241.032,409.428,173.047,32.483,156.003
C01534=1062.290,241.280,409.400,173.049,32.487,156.003
C01535=1062.296,241.528,409.372,173.052,32.491,156.004
C01536=1062.303,241.777,409.344,173.054,32.495,156.005
C01537=1062.309,242.024,409.317,173.057,32.499,156.005
C01538=1062.314,242.274,409.289,173.059,32.503,156.006
C01539=1062.321,242.522,409.262,173.061,32.507,156.007
C01540=1062.326,242.770,409.234,173.064,32.511,156.008
C01541=1062.333,243.019,409.206,173.066,32.515,156.008
C01542=1062.338,243.267,409.178,173.068,32.518,156.009
C01543=1062.345,243.515,409.150,173.070,32.523,156.010
C01544=1062.351,243.764,409.122,173.072,32.526,156.010
C01545=1062.357,244.012,409.095,173.075,32.530,156.011
C01546=1062.363,244.261,409.067,173.077,32.534,156.012
C01547=1062.369,244.509,409.040,173.079,32.538,156.013
C01548=1062.375,244.758,409.011,173.082,32.542,156.013
C01549=1062.381,245.006,408.984,173.084,32.546,156.014
C01550=1062.387,245.254,408.956,173.086,32.550,156.015
C01551=1062.393,245.503,408.927,173.089,32.554,156.016
C01552=1062.399,245.751,408.900,173.091,32.558,156.016
C01553=1062.405,245.999,408.872,173.094,32.562,156.017
C01554=1062.411,246.248,408.844,173.096,32.566,156.018
C01555=1062.417,246.497,408.816,173.098,32.569,156.018
C01556=1062.423,246.745,408.788,173.101,32.574,156.019
C01557=1062.429,246.993,408.760,173.103,32.577,156.020
C01558=1062.435,247.242,408.732,173.106,32.581,156.021
C01559=1062.441,247.489,408.703,173.108,32.585,156.021
C01560=1062.447,247.738,408.675,173.110,32.589,156.022
C01561=1062.454,247.986,408.647,173.113,32.593,156.023
C01562=1062.459,248.235,408.619,173.114,32.597,156.024
C01563=1062.465,248.483,408.591,173.117,32.601,156.024
C01564=1062.471,248.706,408.565,173.119,32.605,156.025
C01565=1062.475,248.929,408.540,173.121,32.608,156.026
C01566=1062.482,249.152,408.514,173.123,32.612,156.026
C01567=1062.487,249.375,408.489,173.125,32.615,156.027
C01568=1062.492,249.598,408.464,173.127,32.619,156.028
C01569=1062.497,249.821,408.439,173.130,32.622,156.028
C01570=1062.503,250.044,408.414,173.132,32.626,156.029
C01571=1062.508,250.267,408.388,173.134,32.629,156.030
C01572=1062.513,250.515,408.360,173.136,32.633,156.030
C01573=1062.520,250.763,408.331,173.139,32.637,156.031
C01574=1062.526,251.012,408.303,173.141,32.641,156.032
C01575=1062.532,251.261,408.275,173.144,32.645,156.033
C01576=1062.538,251.508,408.246,173.146,32.649,156.033
C01577=1062.544,251.757,408.218,173.149,32.653,156.034
C01578=1062.550,252.006,408.189,173.151,32.657,156.035
C01579=1062.557,252.253,408.161,173.154,32.661,156.035
C01580=1062.562,252.501,408.133,173.156,32.665,156.036
C01581=1062.568,252.750,408.105,173.158,32.669,156.037
C01582=1062.574,252.998,408.076,173.161,32.672,156.038
C01583=1062.580,253.247,408.047,173.163,32.677,156.038
C01584=1062.587,253.495,408.018,173.166,32.680,156.039
C01585=1062.593,253.744,407.990,173.168,32.684,156.040
C01586=1062.599,253.992,407.962,173.170,32.688,156.041
C01587=1062.605,254.240,407.933,173.172,32.692,156.041
C01588=1062.611,254.489,407.905,173.175,32.696,156.042
C01589=1062.617,254.737,407.876,173.177,32.700,156.043
C01590=1062.623,254.985,407.848,173.180,32.704,156.043
C01591=1062.629,255.234,407.819,173.182,32.708,156.044
C01592=1062.635,255.481,407.791,173.185,32.712,156.045
C01593=1062.642,255.729,407.762,173.187,32.715,156.046
C01594=1062.647,255.978,407.734,173.190,32.719,156.046
C01595=1062.654,256.226,407.705,173.192,32.723,156.047
C01596=1062.660,256.474,407.676,173.195,32.727,156.048
C01597=1062.666,256.723,407.648,173.197,32.731,156.049
C01598=1062.672,256.971,407.619,173.200,32.735,156.049
C01599=1062.678,257.220,407.590,173.202,32.738,156.050
C01600=1062.685,257.468,407.562,173.205,32.743,156.051
C01601=1062.691,257.716,407.533,173.207,32.746,156.051
C01602=1062.697,257.965,407.504,173.210,32.750,156.052
C01603=1062.703,258.212,407.476,173.212,32.754,156.053
C01604=1062.709,258.460,407.447,173.215,32.758,156.054
C01605=1062.715,258.709,407.418,173.217,32.762,156.054
C01606=1062.721,258.957,407.389,173.220,32.766,156.055
C01607=1062.728,259.205,407.360,173.222,32.770,156.056
C01608=1062.734,259.454,407.332,173.225,32.773,156.056
C01609=1062.740,259.702,407.303,173.228,32.777,156.057
C01610=1062.747,259.950,407.274,173.230,32.781,156.058
C01611=1062.753,260.198,407.245,173.233,32.785,156.059
C01612=1062.759,260.447,407.217,173.235,32.789,156.059
C01613=1062.765,260.695,407.188,173.238,32.793,156.060
C01614=1062.772,260.943,407.159,173.240,32.797,156.061
C01615=1062.778,261.191,407.130,173.243,32.800,156.061
C01616=1062.784,261.439,407.101,173.245,32.804,156.062
C01617=1062.791,261.689,407.072,173.248,32.808,156.063
C01618=1062.797,261.937,407.043,173.251,32.812,156.064
C01619=1062.803,262.185,407.014,173.253,32.816,156.064
C01620=1062.808,262.406,406.989,173.255,32.819,156.065
C01621=1062.814,262.628,406.963,173.257,32.822,156.066
C01622=1062.820,262.851,406.937,173.259,32.826,156.066
C01623=1062.826,263.073,406.911,173.261,32.830,156.067
C01624=1062.832,263.295,406.885,173.264,32.833,156.068
C01625=1062.836,263.516,406.859,173.266,32.836,156.068
C01626=1062.842,263.738,406.833,173.268,32.840,156.069
C01627=1062.848,263.960,406.806,173.270,32.843,156.069
C01628=1062.854,264.208,406.777,173.273,32.847,156.070
C01629=1062.859,264.456,406.748,173.276,32.851,156.071
C01630=1062.866,264.704,406.719,173.278,32.855,156.072
C01631=1062.872,264.953,406.689,173.281,32.859,156.072
C01632=1062.878,265.201,406.660,173.283,32.863,156.073
C01633=1062.884,265.449,406.631,173.286,32.867,156.074
C01634=1062.890,265.697,406.602,173.289,32.871,156.075
C01635=1062.896,265.945,406.573,173.291,32.875,156.075
C01636=1062.902,266.194,406.544,173.294,32.879,156.076
C01637=1062.908,266.442,406.514,173.296,32.883,156.077
C01638=1062.915,266.691,406.485,173.299,32.886,156.078
C01639=1062.921,266.938,406.455,173.302,32.891,156.078
C01640=1062.927,267.187,406.425,173.304,32.894,156.079
C01641=1062.933,267.435,406.396,173.307,32.898,156.080
C01642=1062.939,267.683,406.367,173.309,32.902,156.081
C01643=1062.945,267.931,406.338,173.312,32.906,156.081
C01644=1062.951,268.179,406.308,173.315,32.910,156.082
C01645=1062.958,268.427,406.279,173.317,32.914,156.083
C01646=1062.964,268.676,406.249,173.320,32.918,156.083
C01647=1062.970,268.924,406.220,173.322,32.922,156.084
C01648=1062.977,269.172,406.190,173.325,32.926,156.085
C01649=1062.982,269.420,406.160,173.328,32.930,156.086
C01650=1062.988,269.668,406.131,173.330,32.933,156.086
C01651=1062.994,269.916,406.101,173.333,32.938,156.087
C01652=1063.000,270.164,406.072,173.336,32.941,156.088
C01653=1063.007,270.413,406.042,173.338,32.945,156.089
C01654=1063.013,270.661,406.012,173.341,32.949,156.089
C01655=1063.019,270.909,405.983,173.343,32.953,156.090
C01656=1063.025,271.158,405.953,173.346,32.957,156.091
C01657=1063.031,271.405,405.924,173.349,32.961,156.092
C01658=1063.037,271.654,405.894,173.351,32.965,156.092
C01659=1063.044,271.902,405.864,173.354,32.969,156.093
C01660=1063.050,272.150,405.834,173.357,32.973,156.094
C01661=1063.056,272.398,405.805,173.359,32.977,156.095
C01662=1063.062,272.646,405.775,173.362,32.981,156.095
C01663=1063.069,272.894,405.745,173.365,32.985,156.096
C01664=1063.074,273.143,405.715,173.367,32.988,156.097
C01665=1063.081,273.390,405.685,173.370,32.993,156.098
C01666=1063.086,273.639,405.656,173.373,32.997,156.098
C01667=1063.092,273.887,405.625,173.375,33.000,156.099
C01668=1063.099,274.135,405.596,173.378,33.005,156.100
C01669=1063.105,274.383,405.566,173.381,33.008,156.101
C01670=1063.111,274.631,405.536,173.383,33.013,156.101
C01671=1063.117,274.879,405.506,173.386,33.016,156.102
C01672=1063.123,275.128,405.476,173.389,33.020,156.103
C01673=1063.130,275.375,405.446,173.391,33.024,156.104
C01674=1063.135,275.624,405.416,173.394,33.028,156.104
C01675=1063.141,275.872,405.386,173.397,33.032,156.105
C01676=1063.148,276.095,405.359,173.399,33.036,156.106
C01677=1063.152,276.319,405.332,173.402,33.039,156.107
C01678=1063.158,276.543,405.304,173.404,33.043,156.107
C01679=1063.164,276.766,405.278,173.407,33.047,156.108
C01680=1063.169,276.991,405.251,173.409,33.050,156.108
C01681=1063.174,277.214,405.223,173.411,33.053,156.109
C01682=1063.181,277.438,405.196,173.414,33.057,156.110
C01683=1063.187,277.662,405.169,173.416,33.061,156.111
C01684=1063.192,277.910,405.138,173.419,33.065,156.111
C01685=1063.198,278.158,405.109,173.422,33.069,156.112
C01686=1063.205,278.406,405.078,173.424,33.073,156.113
C01687=1063.211,278.654,405.048,173.427,33.076,156.114
C01688=1063.217,278.902,405.018,173.430,33.081,156.114
C01689=1063.223,279.150,404.987,173.433,33.084,156.115
C01690=1063.230,279.398,404.957,173.435,33.088,156.116
C01691=1063.235,279.646,404.927,173.438,33.092,156.117
C01692=1063.242,279.895,404.897,173.441,33.096,156.117
C01693=1063.247,280.143,404.867,173.445,33.100,156.118
C01694=1063.254,280.390,404.837,173.447,33.104,156.119
C01695=1063.260,280.639,404.806,173.450,33.109,156.120
C01696=1063.266,280.887,404.776,173.453,33.112,156.120
C01697=1063.273,281.135,404.745,173.455,33.116,156.121
C01698=1063.278,281.383,404.715,173.458,33.120,156.122
C01699=1063.284,281.631,404.684,173.461,33.124,156.123
C01700=1063.291,281.879,404.654,173.464,33.129,156.124
C01701=1063.297,282.126,404.623,173.466,33.132,156.124
C01702=1063.303,282.374,404.592,173.469,33.136,156.125
C01703=1063.309,282.623,404.561,173.472,33.141,156.126
C01704=1063.315,282.871,404.531,173.475,33.144,156.127
C01705=1063.321,283.119,404.500,173.477,33.149,156.127
C01706=1063.327,283.367,404.470,173.480,33.152,156.128
C01707=1063.333,283.616,404.439,173.483,33.156,156.129
C01708=1063.339,283.863,404.409,173.486,33.161,156.130
C01709=1063.345,284.111,404.378,173.489,33.164,156.130
C01710=1063.352,284.359,404.347,173.491,33.169,156.131
C01711=1063.358,284.607,404.317,173.494,33.173,156.132
C01712=1063.364,284.855,404.286,173.497,33.176,156.133
C01713=1063.370,285.103,404.256,173.500,33.181,156.133
C01714=1063.377,285.351,404.224,173.502,33.184,156.134
C01715=1063.382,285.599,404.194,173.505,33.189,156.135
C01716=1063.389,285.847,404.163,173.508,33.193,156.136
C01717=1063.395,286.095,404.132,173.511,33.196,156.137
C01718=1063.401,286.343,404.102,173.514,33.201,156.137
C01719=1063.407,286.591,404.071,173.517,33.205,156.138
C01720=1063.414,286.839,404.040,173.519,33.208,156.139
C01721=1063.420,287.087,404.009,173.522,33.213,156.140
C01722=1063.426,287.335,403.979,173.525,33.217,156.140
C01723=1063.433,287.583,403.947,173.528,33.221,156.141
C01724=1063.439,287.831,403.917,173.531,33.225,156.142
C01725=1063.445,288.080,403.886,173.533,33.228,156.143
C01726=1063.451,288.327,403.855,173.537,33.233,156.143
C01727=1063.458,288.575,403.824,173.540,33.237,156.144
C01728=1063.464,288.822,403.793,173.543,33.241,156.145
C01729=1063.470,289.071,403.763,173.546,33.245,156.146
C01730=1063.476,289.319,403.731,173.549,33.249,156.147
C01731=1063.482,289.567,403.700,173.551,33.253,156.147
C01732=1063.488,289.796,403.671,173.554,33.257,156.148
C01733=1063.494,290.025,403.643,173.557,33.261,156.149
C01734=1063.500,290.254,403.614,173.559,33.264,156.150
C01735=1063.505,290.483,403.585,173.562,33.268,156.150
C01736=1063.511,290.712,403.556,173.565,33.272,156.151
C01737=1063.517,290.941,403.528,173.567,33.276,156.152
C01738=1063.522,291.170,403.499,173.570,33.279,156.152
C01739=1063.528,291.399,403.470,173.572,33.283,156.153
C01740=1063.534,291.647,403.438,173.575,33.287,156.154
C01741=1063.540,291.895,403.408,173.578,33.291,156.155
C01742=1063.547,292.143,403.377,173.581,33.295,156.156
C01743=1063.552,292.391,403.345,173.584,33.299,156.156
C01744=1063.559,292.639,403.314,173.587,33.303,156.157
C01745=1063.565,292.887,403.283,173.590,33.308,156.158
C01746=1063.571,293.134,403.252,173.593,33.312,156.159
C01747=1063.577,293.382,403.220,173.595,33.316,156.160
C01748=1063.584,293.631,403.189,173.598,33.320,156.160
C01749=1063.590,293.878,403.158,173.602,33.324,156.161
C01750=1063.596,294.126,403.126,173.605,33.328,156.162
C01751=1063.603,294.374,403.094,173.608,33.332,156.163
C01752=1063.609,294.621,403.063,173.611,33.336,156.164
C01753=1063.615,294.870,403.031,173.614,33.340,156.164
C01754=1063.621,295.118,403.001,173.617,33.344,156.165
C01755=1063.627,295.366,402.969,173.620,33.349,156.166
C01756=1063.633,295.614,402.938,173.622,33.353,156.167
C01757=1063.640,295.861,402.906,173.625,33.357,156.167
C01758=1063.646,296.110,402.874,173.628,33.361,156.168
C01759=1063.652,296.357,402.843,173.631,33.365,156.169
C01760=1063.658,296.605,402.811,173.634,33.369,156.170
C01761=1063.665,296.853,402.780,173.637,33.373,156.171
C01762=1063.671,297.101,402.748,173.640,33.377,156.171
C01763=1063.677,297.348,402.716,173.643,33.382,156.172
C01764=1063.683,297.597,402.684,173.646,33.386,156.173
C01765=1063.689,297.845,402.652,173.650,33.390,156.174
C01766=1063.695,298.092,402.621,173.653,33.394,156.175
C01767=1063.701,298.340,402.589,173.655,33.398,156.176
C01768=1063.707,298.589,402.557,173.658,33.403,156.176
C01769=1063.713,298.837,402.525,173.661,33.407,156.177
C01770=1063.719,299.083,402.493,173.664,33.411,156.178
C01771=1063.725,299.332,402.461,173.667,33.415,156.179
C01772=1063.731,299.580,402.429,173.670,33.419,156.180
C01773=1063.737,299.828,402.397,173.673,33.424,156.180
C01774=1063.744,300.075,402.366,173.676,33.428,156.181
C01775=1063.750,300.323,402.334,173.679,33.432,156.182
C01776=1063.756,300.571,402.302,173.682,33.437,156.183
C01777=1063.762,300.819,402.270,173.685,33.441,156.184
C01778=1063.768,301.066,402.238,173.688,33.445,156.185
C01779=1063.774,301.314,402.206,173.692,33.449,156.186
C01780=1063.780,301.562,402.174,173.695,33.454,156.186
C01781=1063.786,301.810,402.142,173.698,33.458,156.187
C01782=1063.793,302.058,402.110,173.701,33.462,156.188
C01783=1063.799,302.306,402.077,173.704,33.466,156.189
C01784=1063.805,302.553,402.046,173.707,33.470,156.190
C01785=1063.811,302.801,402.013,173.710,33.475,156.190
C01786=1063.818,303.049,401.982,173.713,33.479,156.191
C01787=1063.824,303.296,401.949,173.716,33.483,156.192
C01788=1063.829,303.533,401.918,173.718,33.487,156.193
C01789=1063.835,303.770,401.888,173.721,33.491,156.194
C01790=1063.842,304.007,401.857,173.724,33.495,156.195
C01791=1063.847,304.243,401.826,173.727,33.499,156.195
C01792=1063.853,304.480,401.796,173.731,33.503,156.196
C01793=1063.859,304.716,401.764,173.734,33.508,156.197
C01794=1063.866,304.953,401.734,173.737,33.512,156.198
C01795=1063.871,305.190,401.703,173.740,33.515,156.198
C01796=1063.877,305.438,401.671,173.743,33.520,156.199
C01797=1063.884,305.685,401.638,173.746,33.524,156.200
C01798=1063.890,305.933,401.606,173.749,33.528,156.201
C01799=1063.897,306.181,401.574,173.752,33.533,156.202
C01800=1063.903,306.429,401.542,173.755,33.537,156.203
C01801=1063.909,306.676,401.509,173.758,33.541,156.204
C01802=1063.915,306.924,401.476,173.761,33.545,156.204
C01803=1063.921,307.172,401.444,173.765,33.549,156.205
C01804=1063.928,307.420,401.411,173.768,33.554,156.206
C01805=1063.935,307.667,401.379,173.771,33.558,156.207
C01806=1063.941,307.915,401.347,173.774,33.562,156.208
C01807=1063.947,308.163,401.315,173.777,33.567,156.209
C01808=1063.953,308.411,401.282,173.780,33.571,156.209
C01809=1063.959,308.659,401.250,173.783,33.575,156.210
C01810=1063.965,308.906,401.217,173.786,33.579,156.211
C01811=1063.972,309.154,401.184,173.789,33.583,156.212
C01812=1063.979,309.401,401.152,173.792,33.588,156.213
C01813=1063.985,309.649,401.119,173.796,33.592,156.214
C01814=1063.991,309.897,401.087,173.800,33.597,156.214
